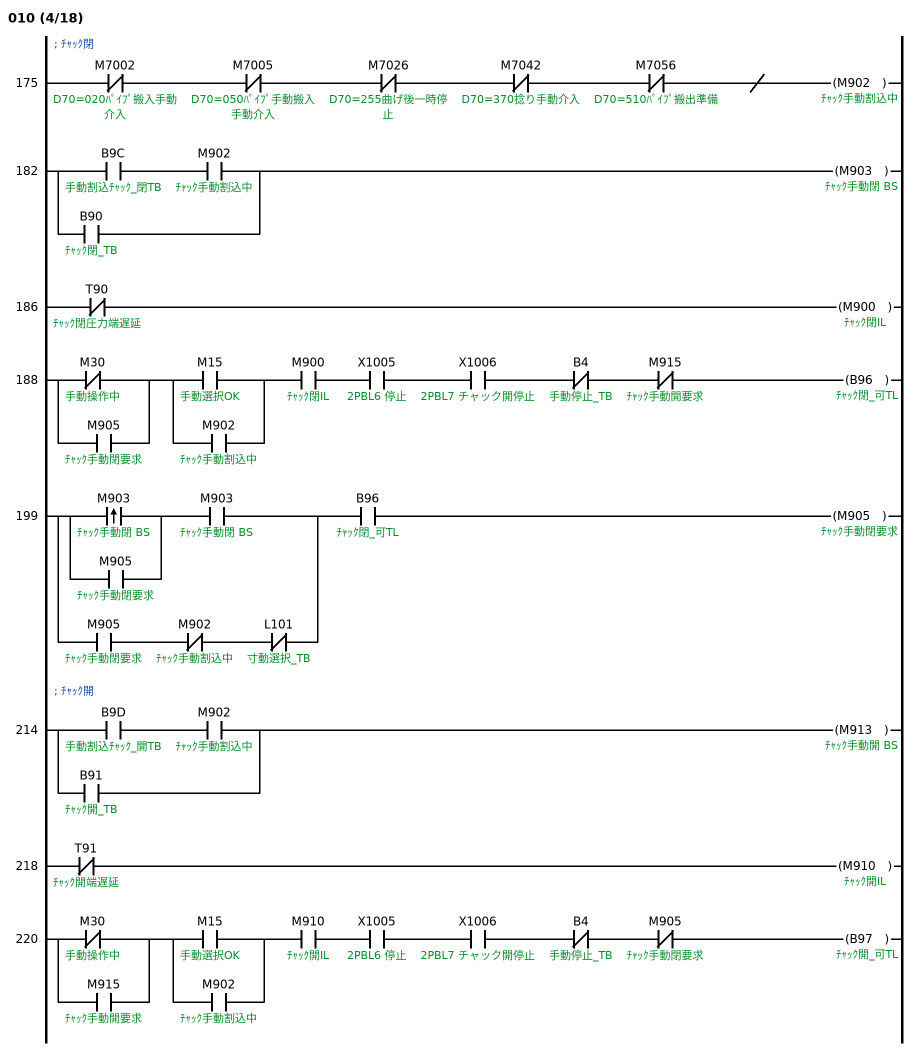
; ﾁｬｯｸ閉
175   LDI     M7002  ; D70=020ﾊﾟｲﾌﾟ搬入手動介入
      ANI     M7005  ; D70=050ﾊﾟｲﾌﾟ手動搬入手動介入
      ANI     M7026  ; D70=255曲げ後一時停止
      ANI     M7042  ; D70=370捻り手動介入
      ANI     M7056  ; D70=510ﾊﾟｲﾌﾟ搬出準備
      INV
      OUT     M902  ; ﾁｬｯｸ手動割込中
182   LD      B9C  ; 手動割込ﾁｬｯｸ_閉TB
      AND     M902  ; ﾁｬｯｸ手動割込中
      OR      B90  ; ﾁｬｯｸ閉_TB
      OUT     M903  ; ﾁｬｯｸ手動閉 BS
186   LDI     T90  ; ﾁｬｯｸ閉圧力端遅延
      OUT     M900  ; ﾁｬｯｸ閉IL
188   LDI     M30  ; 手動操作中
      OR      M905  ; ﾁｬｯｸ手動閉要求
      LD      M15  ; 手動選択OK
      OR      M902  ; ﾁｬｯｸ手動割込中
      ANB
      AND     M900  ; ﾁｬｯｸ閉IL
      AND     X1005  ; 2PBL6 停止
      AND     X1006  ; 2PBL7 チャック開停止
      ANI     B4  ; 手動停止_TB
      ANI     M915  ; ﾁｬｯｸ手動開要求
      OUT     B96  ; ﾁｬｯｸ閉_可TL
199   LDP     M903  ; ﾁｬｯｸ手動閉 BS
      OR      M905  ; ﾁｬｯｸ手動閉要求
      AND     M903  ; ﾁｬｯｸ手動閉 BS
      LD      M905  ; ﾁｬｯｸ手動閉要求
      ANI     M902  ; ﾁｬｯｸ手動割込中
      ANI     L101  ; 寸動選択_TB
      ORB
      AND     B96  ; ﾁｬｯｸ閉_可TL
      OUT     M905  ; ﾁｬｯｸ手動閉要求
; ﾁｬｯｸ開
214   LD      B9D  ; 手動割込ﾁｬｯｸ_開TB
      AND     M902  ; ﾁｬｯｸ手動割込中
      OR      B91  ; ﾁｬｯｸ開_TB
      OUT     M913  ; ﾁｬｯｸ手動開 BS
218   LDI     T91  ; ﾁｬｯｸ開端遅延
      OUT     M910  ; ﾁｬｯｸ開IL
220   LDI     M30  ; 手動操作中
      OR      M915  ; ﾁｬｯｸ手動開要求
      LD      M15  ; 手動選択OK
      OR      M902  ; ﾁｬｯｸ手動割込中
      ANB
      AND     M910  ; ﾁｬｯｸ開IL
      AND     X1005  ; 2PBL6 停止
      AND     X1006  ; 2PBL7 チャック開停止
      ANI     B4  ; 手動停止_TB
      ANI     M905  ; ﾁｬｯｸ手動閉要求
      OUT     B97  ; ﾁｬｯｸ開_可TL
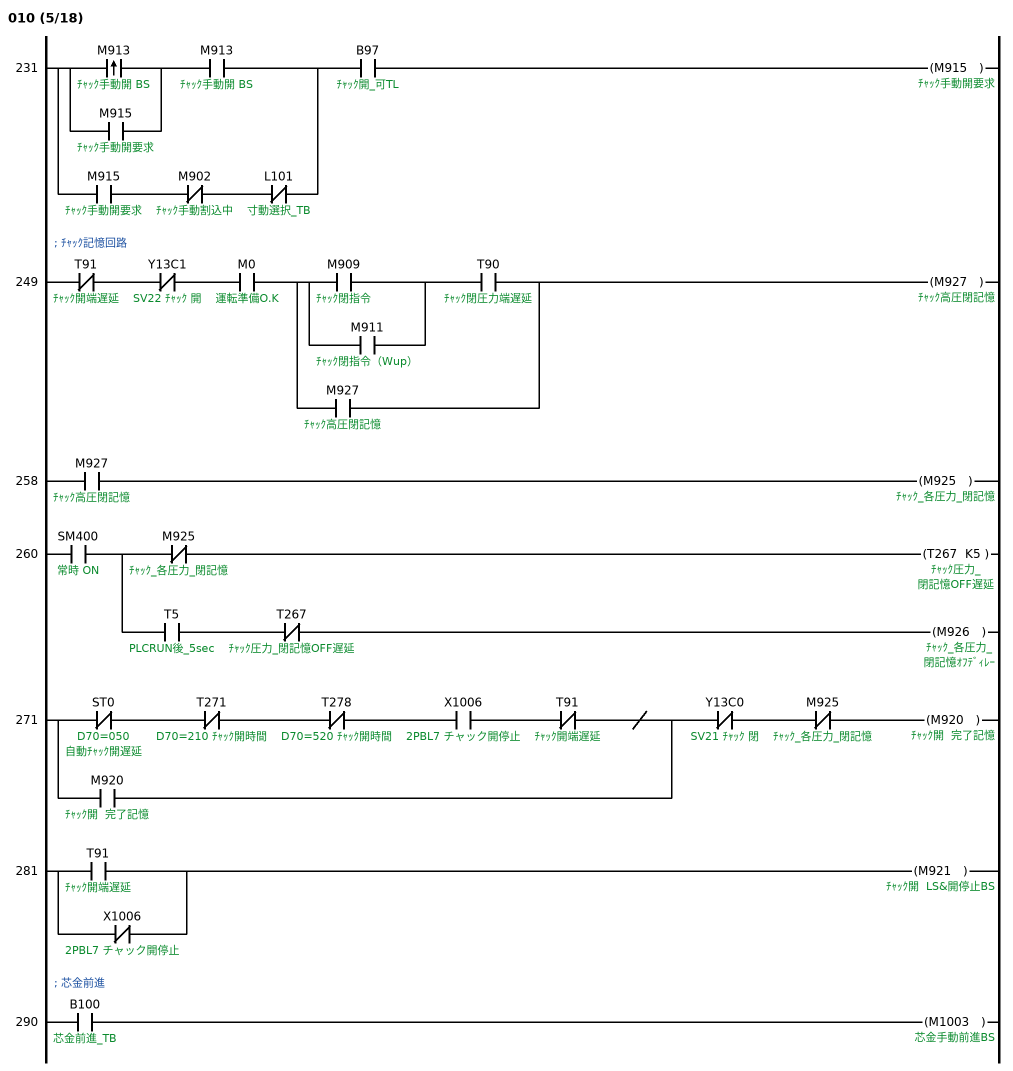
231   LDP     M913  ; ﾁｬｯｸ手動開 BS
      OR      M915  ; ﾁｬｯｸ手動開要求
      AND     M913  ; ﾁｬｯｸ手動開 BS
      LD      M915  ; ﾁｬｯｸ手動開要求
      ANI     M902  ; ﾁｬｯｸ手動割込中
      ANI     L101  ; 寸動選択_TB
      ORB
      AND     B97  ; ﾁｬｯｸ開_可TL
      OUT     M915  ; ﾁｬｯｸ手動開要求
; ﾁｬｯｸ記憶回路
249   LDI     T91  ; ﾁｬｯｸ開端遅延
      ANI     Y13C1  ; SV22 ﾁｬｯｸ 開
      AND     M0  ; 運転準備O.K
      LD      M909  ; ﾁｬｯｸ閉指令
      OR      M911  ; ﾁｬｯｸ閉指令（Wup）
      AND     T90  ; ﾁｬｯｸ閉圧力端遅延
      OR      M927  ; ﾁｬｯｸ高圧閉記憶
      ANB
      OUT     M927  ; ﾁｬｯｸ高圧閉記憶
258   LD      M927  ; ﾁｬｯｸ高圧閉記憶
      OUT     M925  ; ﾁｬｯｸ_各圧力_閉記憶
260   LD      SM400  ; 常時 ON
      MPS
      ANI     M925  ; ﾁｬｯｸ_各圧力_閉記憶
      OUT     T267 K5  ; ﾁｬｯｸ圧力_閉記憶OFF遅延
      MPP
      AND     T5  ; PLCRUN後_5sec
      ANI     T267  ; ﾁｬｯｸ圧力_閉記憶OFF遅延
      OUT     M926  ; ﾁｬｯｸ_各圧力_閉記憶ｵﾌﾃﾞｨﾚｰ
271   LDI     ST0  ; D70=050 自動ﾁｬｯｸ開遅延
      ANI     T271  ; D70=210 ﾁｬｯｸ開時間
      ANI     T278  ; D70=520 ﾁｬｯｸ開時間
      AND     X1006  ; 2PBL7 チャック開停止
      ANI     T91  ; ﾁｬｯｸ開端遅延
      INV
      OR      M920  ; ﾁｬｯｸ開  完了記憶
      ANI     Y13C0  ; SV21 ﾁｬｯｸ 閉
      ANI     M925  ; ﾁｬｯｸ_各圧力_閉記憶
      OUT     M920  ; ﾁｬｯｸ開  完了記憶
281   LD      T91  ; ﾁｬｯｸ開端遅延
      ORI     X1006  ; 2PBL7 チャック開停止
      OUT     M921  ; ﾁｬｯｸ開  LS&開停止BS
; 芯金前進
290   LD      B100  ; 芯金前進_TB
      OUT     M1003  ; 芯金手動前進BS
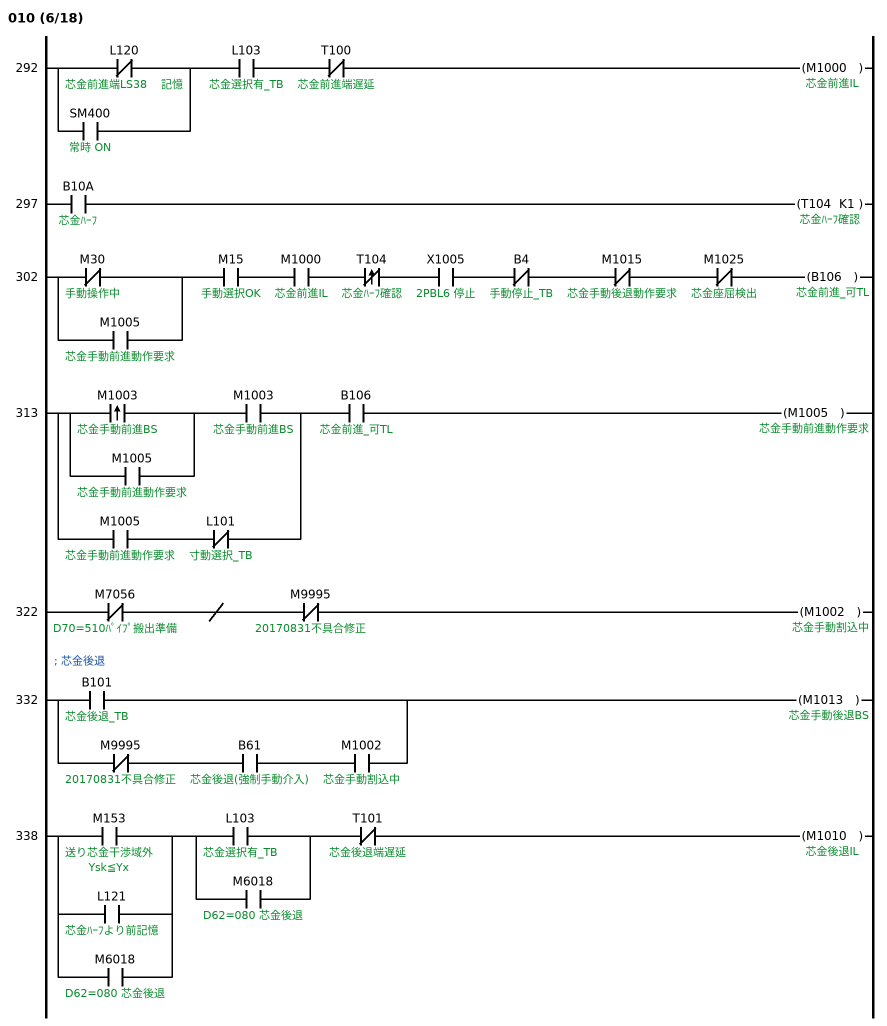
292   LDI     L120  ; 芯金前進端LS38    記憶
      OR      SM400  ; 常時 ON
      AND     L103  ; 芯金選択有_TB
      ANI     T100  ; 芯金前進端遅延
      OUT     M1000  ; 芯金前進IL
297   LD      B10A  ; 芯金ﾊｰﾌ
      OUT     T104 K1  ; 芯金ﾊｰﾌ確認
302   LDI     M30  ; 手動操作中
      OR      M1005  ; 芯金手動前進動作要求
      AND     M15  ; 手動選択OK
      AND     M1000  ; 芯金前進IL
      ANDPI   T104  ; 芯金ﾊｰﾌ確認
      AND     X1005  ; 2PBL6 停止
      ANI     B4  ; 手動停止_TB
      ANI     M1015  ; 芯金手動後退動作要求
      ANI     M1025  ; 芯金座屈検出
      OUT     B106  ; 芯金前進_可TL
313   LDP     M1003  ; 芯金手動前進BS
      OR      M1005  ; 芯金手動前進動作要求
      AND     M1003  ; 芯金手動前進BS
      LD      M1005  ; 芯金手動前進動作要求
      ANI     L101  ; 寸動選択_TB
      ORB
      AND     B106  ; 芯金前進_可TL
      OUT     M1005  ; 芯金手動前進動作要求
322   LDI     M7056  ; D70=510ﾊﾟｲﾌﾟ搬出準備
      INV
      ANI     M9995  ; 20170831不具合修正
      OUT     M1002  ; 芯金手動割込中
; 芯金後退
332   LD      B101  ; 芯金後退_TB
      LDI     M9995  ; 20170831不具合修正
      AND     B61  ; 芯金後退(強制手動介入)
      AND     M1002  ; 芯金手動割込中
      ORB
      OUT     M1013  ; 芯金手動後退BS
338   LD      M153  ; 送り芯金干渉域外 Ysk≦Yx
      OR      L121  ; 芯金ﾊｰﾌより前記憶
      OR      M6018  ; D62=080 芯金後退
      LD      L103  ; 芯金選択有_TB
      OR      M6018  ; D62=080 芯金後退
      ANB
      ANI     T101  ; 芯金後退端遅延
      OUT     M1010  ; 芯金後退IL
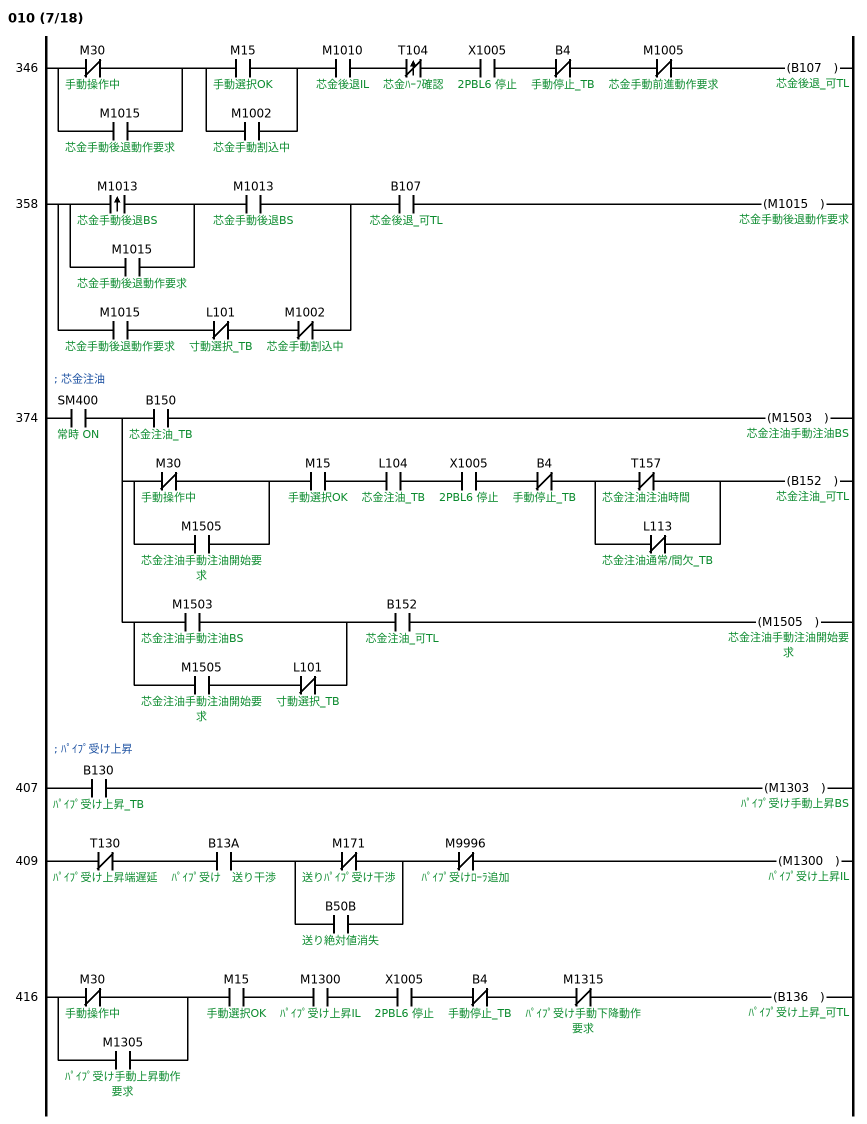
346   LDI     M30  ; 手動操作中
      OR      M1015  ; 芯金手動後退動作要求
      LD      M15  ; 手動選択OK
      OR      M1002  ; 芯金手動割込中
      ANB
      AND     M1010  ; 芯金後退IL
      ANDPI   T104  ; 芯金ﾊｰﾌ確認
      AND     X1005  ; 2PBL6 停止
      ANI     B4  ; 手動停止_TB
      ANI     M1005  ; 芯金手動前進動作要求
      OUT     B107  ; 芯金後退_可TL
358   LDP     M1013  ; 芯金手動後退BS
      OR      M1015  ; 芯金手動後退動作要求
      AND     M1013  ; 芯金手動後退BS
      LD      M1015  ; 芯金手動後退動作要求
      ANI     L101  ; 寸動選択_TB
      ANI     M1002  ; 芯金手動割込中
      ORB
      AND     B107  ; 芯金後退_可TL
      OUT     M1015  ; 芯金手動後退動作要求
; 芯金注油
374   LD      SM400  ; 常時 ON
      MPS
      AND     B150  ; 芯金注油_TB
      OUT     M1503  ; 芯金注油手動注油BS
      MRD
      LDI     M30  ; 手動操作中
      OR      M1505  ; 芯金注油手動注油開始要求
      ANB
      AND     M15  ; 手動選択OK
      AND     L104  ; 芯金注油_TB
      AND     X1005  ; 2PBL6 停止
      ANI     B4  ; 手動停止_TB
      LDI     T157  ; 芯金注油注油時間
      ORI     L113  ; 芯金注油通常/間欠_TB
      ANB
      OUT     B152  ; 芯金注油_可TL
      MPP
      LD      M1503  ; 芯金注油手動注油BS
      LD      M1505  ; 芯金注油手動注油開始要求
      ANI     L101  ; 寸動選択_TB
      ORB
      ANB
      AND     B152  ; 芯金注油_可TL
      OUT     M1505  ; 芯金注油手動注油開始要求
; ﾊﾟｲﾌﾟ受け上昇
407   LD      B130  ; ﾊﾟｲﾌﾟ受け上昇_TB
      OUT     M1303  ; ﾊﾟｲﾌﾟ受け手動上昇BS
409   LDI     T130  ; ﾊﾟｲﾌﾟ受け上昇端遅延
      AND     B13A  ; ﾊﾟｲﾌﾟ受け　送り干渉
      LDI     M171  ; 送りﾊﾟｲﾌﾟ受け干渉
      OR      B50B  ; 送り絶対値消失
      ANB
      ANI     M9996  ; ﾊﾟｲﾌﾟ受けﾛｰﾗ追加
      OUT     M1300  ; ﾊﾟｲﾌﾟ受け上昇IL
416   LDI     M30  ; 手動操作中
      OR      M1305  ; ﾊﾟｲﾌﾟ受け手動上昇動作要求
      AND     M15  ; 手動選択OK
      AND     M1300  ; ﾊﾟｲﾌﾟ受け上昇IL
      AND     X1005  ; 2PBL6 停止
      ANI     B4  ; 手動停止_TB
      ANI     M1315  ; ﾊﾟｲﾌﾟ受け手動下降動作要求
      OUT     B136  ; ﾊﾟｲﾌﾟ受け上昇_可TL
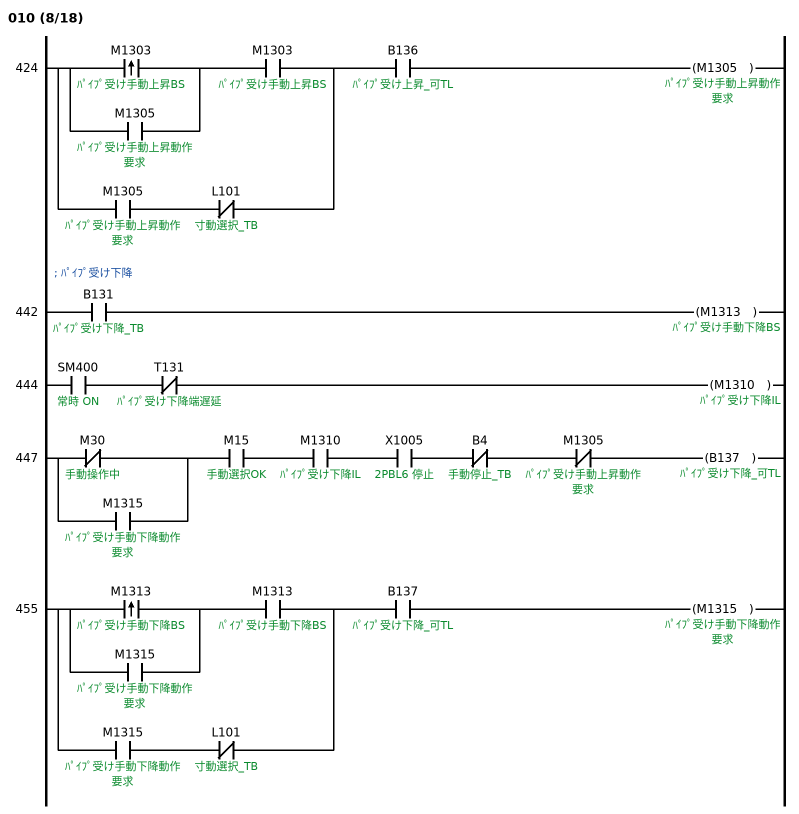
424   LDP     M1303  ; ﾊﾟｲﾌﾟ受け手動上昇BS
      OR      M1305  ; ﾊﾟｲﾌﾟ受け手動上昇動作要求
      AND     M1303  ; ﾊﾟｲﾌﾟ受け手動上昇BS
      LD      M1305  ; ﾊﾟｲﾌﾟ受け手動上昇動作要求
      ANI     L101  ; 寸動選択_TB
      ORB
      AND     B136  ; ﾊﾟｲﾌﾟ受け上昇_可TL
      OUT     M1305  ; ﾊﾟｲﾌﾟ受け手動上昇動作要求
; ﾊﾟｲﾌﾟ受け下降
442   LD      B131  ; ﾊﾟｲﾌﾟ受け下降_TB
      OUT     M1313  ; ﾊﾟｲﾌﾟ受け手動下降BS
444   LD      SM400  ; 常時 ON
      ANI     T131  ; ﾊﾟｲﾌﾟ受け下降端遅延
      OUT     M1310  ; ﾊﾟｲﾌﾟ受け下降IL
447   LDI     M30  ; 手動操作中
      OR      M1315  ; ﾊﾟｲﾌﾟ受け手動下降動作要求
      AND     M15  ; 手動選択OK
      AND     M1310  ; ﾊﾟｲﾌﾟ受け下降IL
      AND     X1005  ; 2PBL6 停止
      ANI     B4  ; 手動停止_TB
      ANI     M1305  ; ﾊﾟｲﾌﾟ受け手動上昇動作要求
      OUT     B137  ; ﾊﾟｲﾌﾟ受け下降_可TL
455   LDP     M1313  ; ﾊﾟｲﾌﾟ受け手動下降BS
      OR      M1315  ; ﾊﾟｲﾌﾟ受け手動下降動作要求
      AND     M1313  ; ﾊﾟｲﾌﾟ受け手動下降BS
      LD      M1315  ; ﾊﾟｲﾌﾟ受け手動下降動作要求
      ANI     L101  ; 寸動選択_TB
      ORB
      AND     B137  ; ﾊﾟｲﾌﾟ受け下降_可TL
      OUT     M1315  ; ﾊﾟｲﾌﾟ受け手動下降動作要求
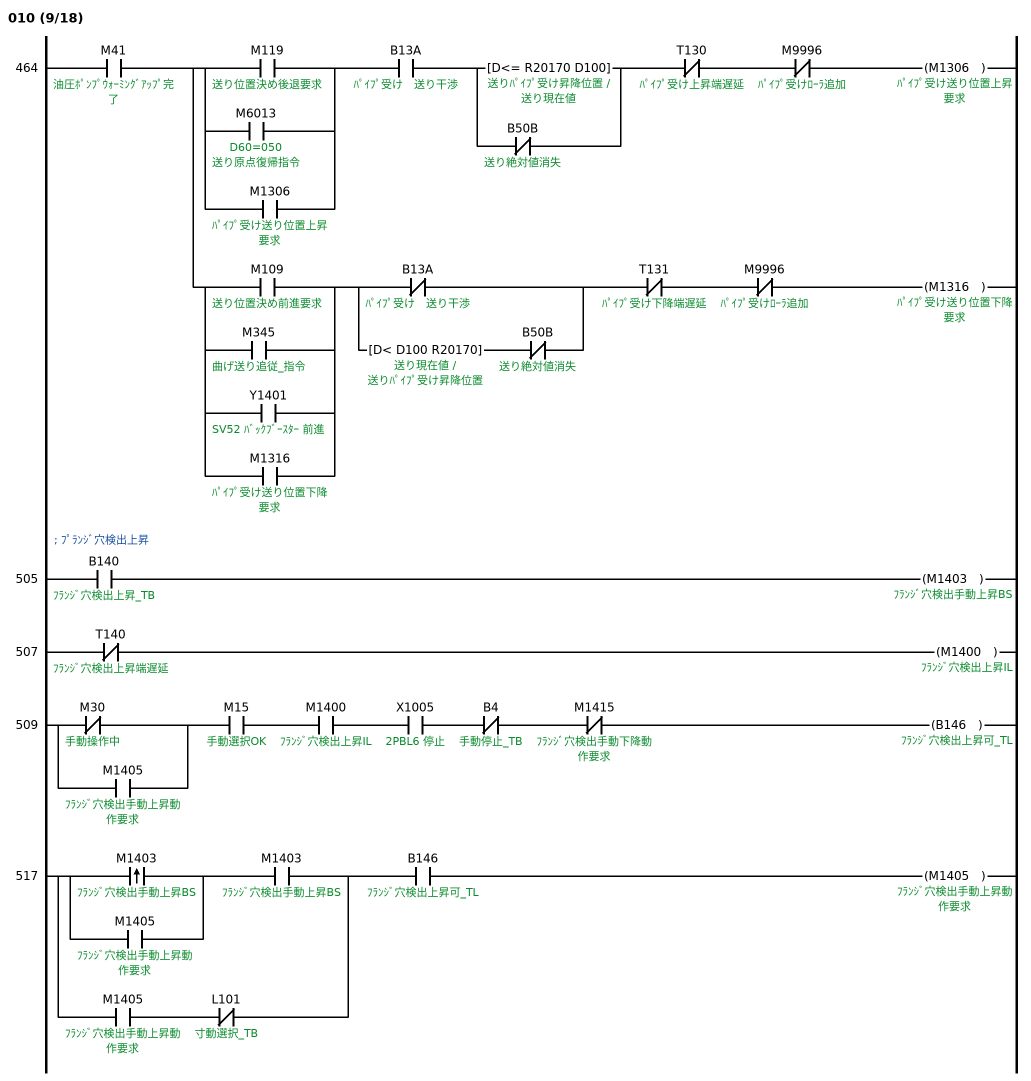
464   LD      M41  ; 油圧ﾎﾟﾝﾌﾟｳｫｰﾐﾝｸﾞｱｯﾌﾟ完了
      MPS
      LD      M119  ; 送り位置決め後退要求
      OR      M6013  ; D60=050 送り原点復帰指令
      OR      M1306  ; ﾊﾟｲﾌﾟ受け送り位置上昇要求
      ANB
      AND     B13A  ; ﾊﾟｲﾌﾟ受け　送り干渉
      LDD<=   R20170 D100  ; 送りﾊﾟｲﾌﾟ受け昇降位置 / 送り現在値
      ORI     B50B  ; 送り絶対値消失
      ANB
      ANI     T130  ; ﾊﾟｲﾌﾟ受け上昇端遅延
      ANI     M9996  ; ﾊﾟｲﾌﾟ受けﾛｰﾗ追加
      OUT     M1306  ; ﾊﾟｲﾌﾟ受け送り位置上昇要求
      MPP
      LD      M109  ; 送り位置決め前進要求
      OR      M345  ; 曲げ送り追従_指令
      OR      Y1401  ; SV52 ﾊﾞｯｸﾌﾞｰｽﾀｰ 前進
      OR      M1316  ; ﾊﾟｲﾌﾟ受け送り位置下降要求
      ANB
      LDI     B13A  ; ﾊﾟｲﾌﾟ受け　送り干渉
      LDD<    D100 R20170  ; 送り現在値 / 送りﾊﾟｲﾌﾟ受け昇降位置
      ANI     B50B  ; 送り絶対値消失
      ORB
      ANB
      ANI     T131  ; ﾊﾟｲﾌﾟ受け下降端遅延
      ANI     M9996  ; ﾊﾟｲﾌﾟ受けﾛｰﾗ追加
      OUT     M1316  ; ﾊﾟｲﾌﾟ受け送り位置下降要求
; ﾌﾟﾗﾝｼﾞ穴検出上昇
505   LD      B140  ; ﾌﾗﾝｼﾞ穴検出上昇_TB
      OUT     M1403  ; ﾌﾗﾝｼﾞ穴検出手動上昇BS
507   LDI     T140  ; ﾌﾗﾝｼﾞ穴検出上昇端遅延
      OUT     M1400  ; ﾌﾗﾝｼﾞ穴検出上昇IL
509   LDI     M30  ; 手動操作中
      OR      M1405  ; ﾌﾗﾝｼﾞ穴検出手動上昇動作要求
      AND     M15  ; 手動選択OK
      AND     M1400  ; ﾌﾗﾝｼﾞ穴検出上昇IL
      AND     X1005  ; 2PBL6 停止
      ANI     B4  ; 手動停止_TB
      ANI     M1415  ; ﾌﾗﾝｼﾞ穴検出手動下降動作要求
      OUT     B146  ; ﾌﾗﾝｼﾞ穴検出上昇可_TL
517   LDP     M1403  ; ﾌﾗﾝｼﾞ穴検出手動上昇BS
      OR      M1405  ; ﾌﾗﾝｼﾞ穴検出手動上昇動作要求
      AND     M1403  ; ﾌﾗﾝｼﾞ穴検出手動上昇BS
      LD      M1405  ; ﾌﾗﾝｼﾞ穴検出手動上昇動作要求
      ANI     L101  ; 寸動選択_TB
      ORB
      AND     B146  ; ﾌﾗﾝｼﾞ穴検出上昇可_TL
      OUT     M1405  ; ﾌﾗﾝｼﾞ穴検出手動上昇動作要求
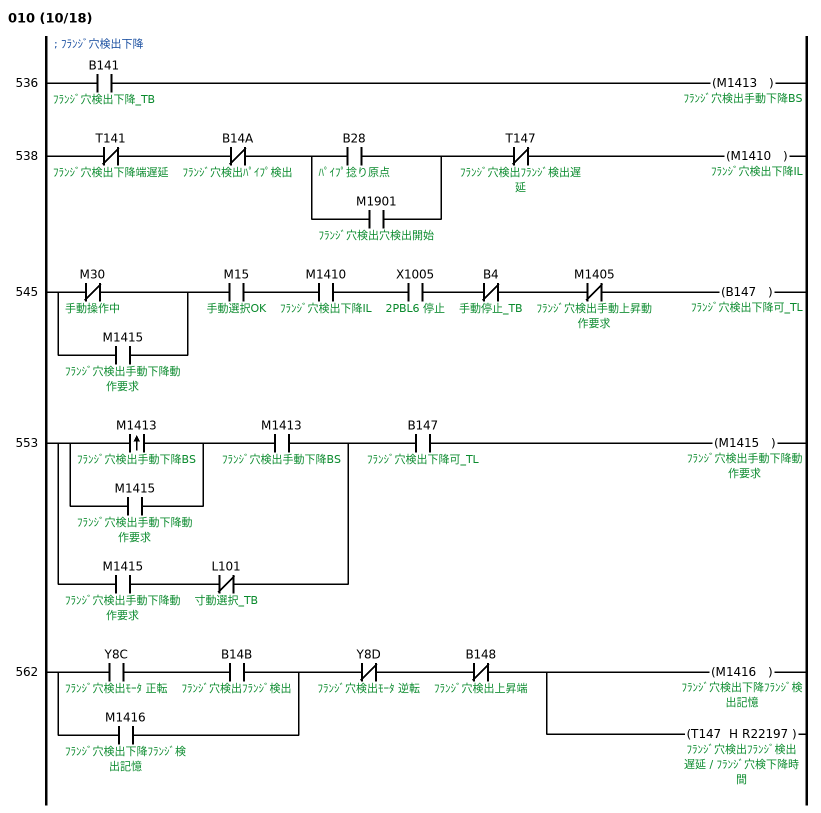
; ﾌﾗﾝｼﾞ穴検出下降
536   LD      B141  ; ﾌﾗﾝｼﾞ穴検出下降_TB
      OUT     M1413  ; ﾌﾗﾝｼﾞ穴検出手動下降BS
538   LDI     T141  ; ﾌﾗﾝｼﾞ穴検出下降端遅延
      ANI     B14A  ; ﾌﾗﾝｼﾞ穴検出ﾊﾟｲﾌﾟ検出
      LD      B28  ; ﾊﾟｲﾌﾟ捻り原点
      OR      M1901  ; ﾌﾗﾝｼﾞ穴検出穴検出開始
      ANB
      ANI     T147  ; ﾌﾗﾝｼﾞ穴検出ﾌﾗﾝｼﾞ検出遅延
      OUT     M1410  ; ﾌﾗﾝｼﾞ穴検出下降IL
545   LDI     M30  ; 手動操作中
      OR      M1415  ; ﾌﾗﾝｼﾞ穴検出手動下降動作要求
      AND     M15  ; 手動選択OK
      AND     M1410  ; ﾌﾗﾝｼﾞ穴検出下降IL
      AND     X1005  ; 2PBL6 停止
      ANI     B4  ; 手動停止_TB
      ANI     M1405  ; ﾌﾗﾝｼﾞ穴検出手動上昇動作要求
      OUT     B147  ; ﾌﾗﾝｼﾞ穴検出下降可_TL
553   LDP     M1413  ; ﾌﾗﾝｼﾞ穴検出手動下降BS
      OR      M1415  ; ﾌﾗﾝｼﾞ穴検出手動下降動作要求
      AND     M1413  ; ﾌﾗﾝｼﾞ穴検出手動下降BS
      LD      M1415  ; ﾌﾗﾝｼﾞ穴検出手動下降動作要求
      ANI     L101  ; 寸動選択_TB
      ORB
      AND     B147  ; ﾌﾗﾝｼﾞ穴検出下降可_TL
      OUT     M1415  ; ﾌﾗﾝｼﾞ穴検出手動下降動作要求
562   LD      Y8C  ; ﾌﾗﾝｼﾞ穴検出ﾓｰﾀ 正転
      AND     B14B  ; ﾌﾗﾝｼﾞ穴検出ﾌﾗﾝｼﾞ検出
      OR      M1416  ; ﾌﾗﾝｼﾞ穴検出下降ﾌﾗﾝｼﾞ検出記憶
      ANI     Y8D  ; ﾌﾗﾝｼﾞ穴検出ﾓｰﾀ 逆転
      ANI     B148  ; ﾌﾗﾝｼﾞ穴検出上昇端
      OUT     M1416  ; ﾌﾗﾝｼﾞ穴検出下降ﾌﾗﾝｼﾞ検出記憶
      OUTH    T147 R22197  ; ﾌﾗﾝｼﾞ穴検出ﾌﾗﾝｼﾞ検出遅延 / ﾌﾗﾝｼﾞ穴検下降時間
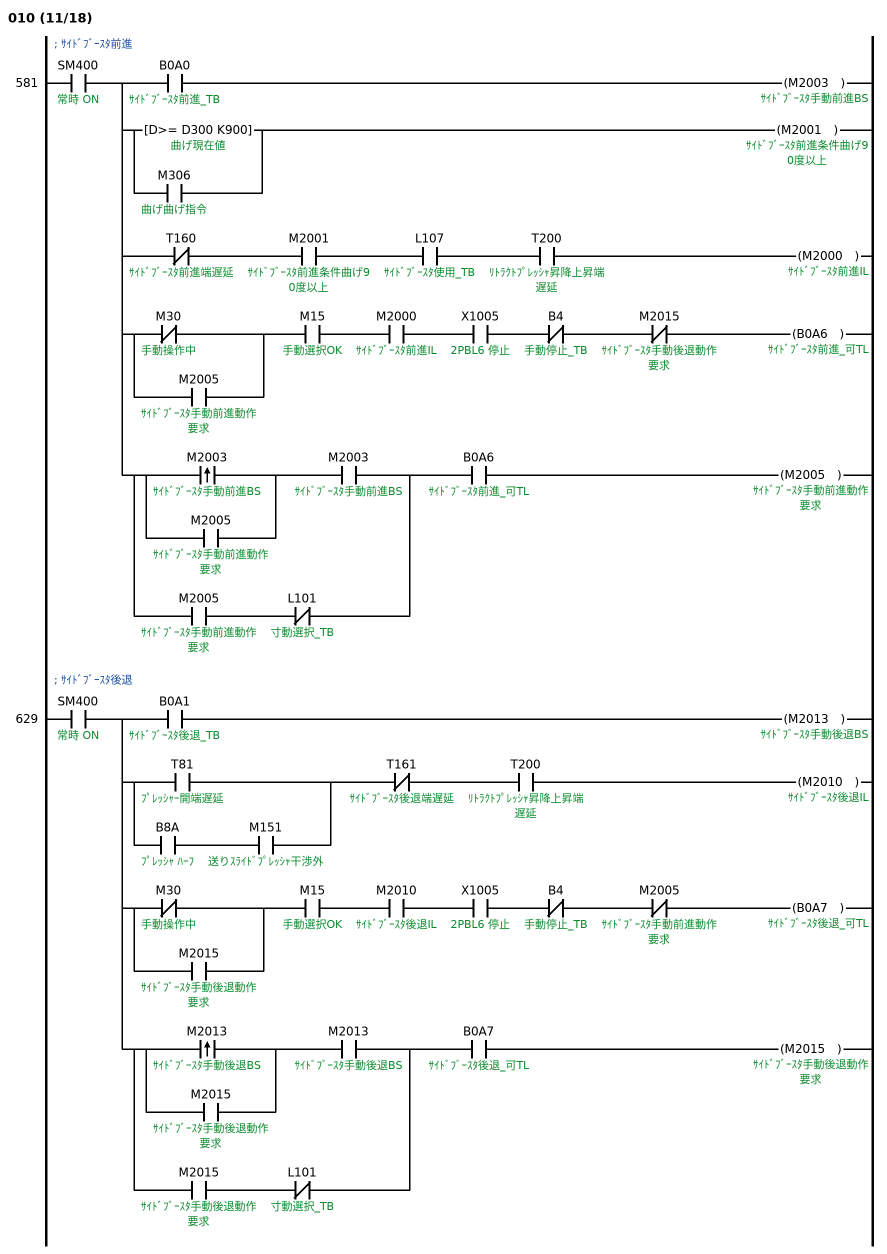
; ｻｲﾄﾞﾌﾞｰｽﾀ前進
581   LD      SM400  ; 常時 ON
      MPS
      AND     B0A0  ; ｻｲﾄﾞﾌﾞｰｽﾀ前進_TB
      OUT     M2003  ; ｻｲﾄﾞﾌﾞｰｽﾀ手動前進BS
      MRD
      LDD>=   D300 K900  ; 曲げ現在値
      OR      M306  ; 曲げ曲げ指令
      ANB
      OUT     M2001  ; ｻｲﾄﾞﾌﾞｰｽﾀ前進条件曲げ90度以上
      MRD
      ANI     T160  ; ｻｲﾄﾞﾌﾞｰｽﾀ前進端遅延
      AND     M2001  ; ｻｲﾄﾞﾌﾞｰｽﾀ前進条件曲げ90度以上
      AND     L107  ; ｻｲﾄﾞﾌﾞｰｽﾀ使用_TB
      AND     T200  ; ﾘﾄﾗｸﾄﾌﾟﾚｯｼｬ昇降上昇端遅延
      OUT     M2000  ; ｻｲﾄﾞﾌﾞｰｽﾀ前進IL
      MRD
      LDI     M30  ; 手動操作中
      OR      M2005  ; ｻｲﾄﾞﾌﾞｰｽﾀ手動前進動作要求
      ANB
      AND     M15  ; 手動選択OK
      AND     M2000  ; ｻｲﾄﾞﾌﾞｰｽﾀ前進IL
      AND     X1005  ; 2PBL6 停止
      ANI     B4  ; 手動停止_TB
      ANI     M2015  ; ｻｲﾄﾞﾌﾞｰｽﾀ手動後退動作要求
      OUT     B0A6  ; ｻｲﾄﾞﾌﾞｰｽﾀ前進_可TL
      MPP
      LDP     M2003  ; ｻｲﾄﾞﾌﾞｰｽﾀ手動前進BS
      OR      M2005  ; ｻｲﾄﾞﾌﾞｰｽﾀ手動前進動作要求
      AND     M2003  ; ｻｲﾄﾞﾌﾞｰｽﾀ手動前進BS
      LD      M2005  ; ｻｲﾄﾞﾌﾞｰｽﾀ手動前進動作要求
      ANI     L101  ; 寸動選択_TB
      ORB
      ANB
      AND     B0A6  ; ｻｲﾄﾞﾌﾞｰｽﾀ前進_可TL
      OUT     M2005  ; ｻｲﾄﾞﾌﾞｰｽﾀ手動前進動作要求
; ｻｲﾄﾞﾌﾞｰｽﾀ後退
629   LD      SM400  ; 常時 ON
      MPS
      AND     B0A1  ; ｻｲﾄﾞﾌﾞｰｽﾀ後退_TB
      OUT     M2013  ; ｻｲﾄﾞﾌﾞｰｽﾀ手動後退BS
      MRD
      LD      T81  ; ﾌﾟﾚｯｼｬｰ開端遅延
      LD      B8A  ; ﾌﾟﾚｯｼｬ ﾊｰﾌ
      AND     M151  ; 送りｽﾗｲﾄﾞﾌﾟﾚｯｼｬ干渉外
      ORB
      ANB
      ANI     T161  ; ｻｲﾄﾞﾌﾞｰｽﾀ後退端遅延
      AND     T200  ; ﾘﾄﾗｸﾄﾌﾟﾚｯｼｬ昇降上昇端遅延
      OUT     M2010  ; ｻｲﾄﾞﾌﾞｰｽﾀ後退IL
      MRD
      LDI     M30  ; 手動操作中
      OR      M2015  ; ｻｲﾄﾞﾌﾞｰｽﾀ手動後退動作要求
      ANB
      AND     M15  ; 手動選択OK
      AND     M2010  ; ｻｲﾄﾞﾌﾞｰｽﾀ後退IL
      AND     X1005  ; 2PBL6 停止
      ANI     B4  ; 手動停止_TB
      ANI     M2005  ; ｻｲﾄﾞﾌﾞｰｽﾀ手動前進動作要求
      OUT     B0A7  ; ｻｲﾄﾞﾌﾞｰｽﾀ後退_可TL
      MPP
      LDP     M2013  ; ｻｲﾄﾞﾌﾞｰｽﾀ手動後退BS
      OR      M2015  ; ｻｲﾄﾞﾌﾞｰｽﾀ手動後退動作要求
      AND     M2013  ; ｻｲﾄﾞﾌﾞｰｽﾀ手動後退BS
      LD      M2015  ; ｻｲﾄﾞﾌﾞｰｽﾀ手動後退動作要求
      ANI     L101  ; 寸動選択_TB
      ORB
      ANB
      AND     B0A7  ; ｻｲﾄﾞﾌﾞｰｽﾀ後退_可TL
      OUT     M2015  ; ｻｲﾄﾞﾌﾞｰｽﾀ手動後退動作要求
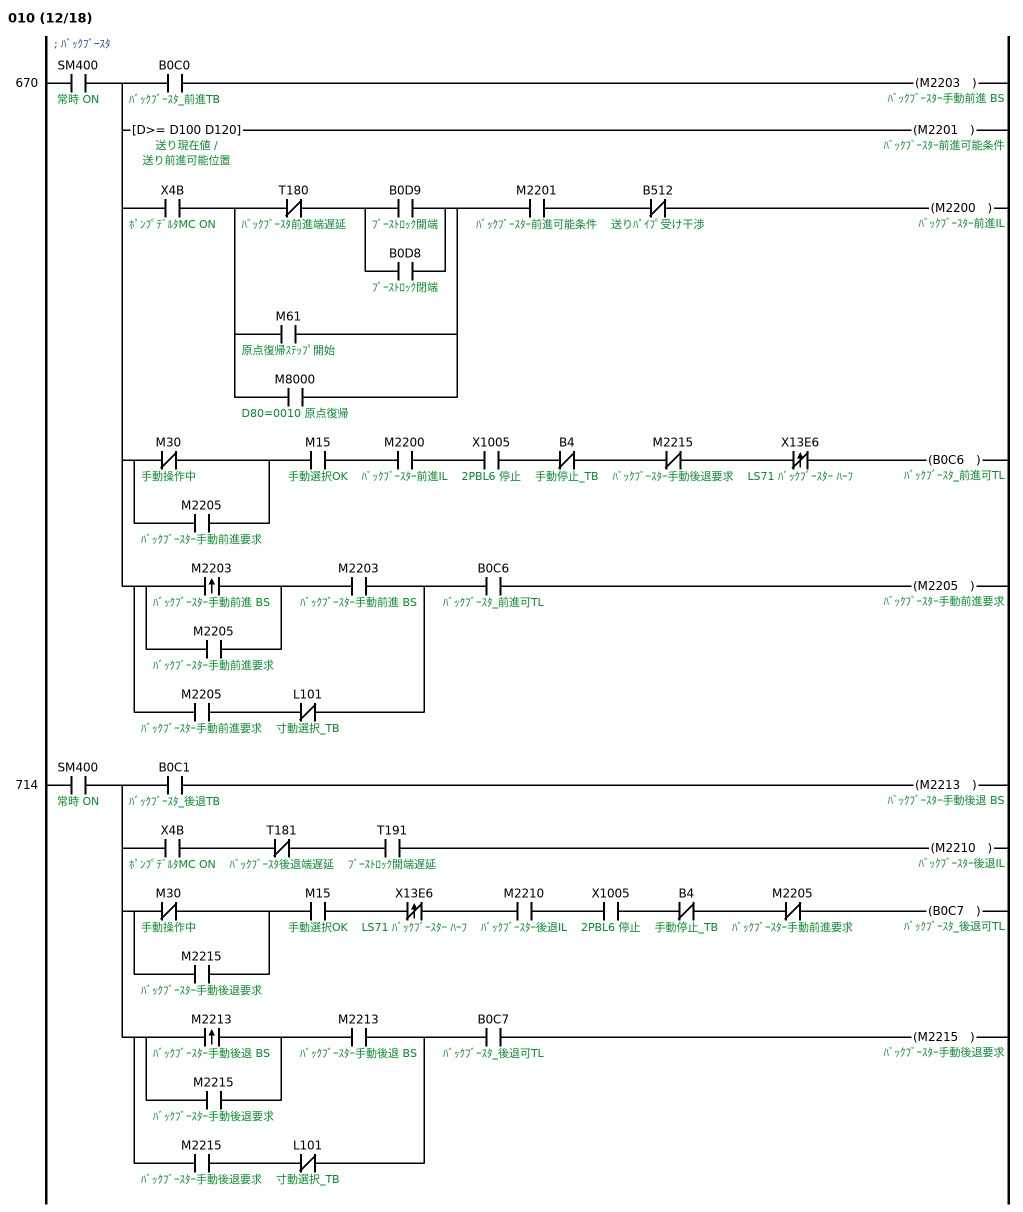
; ﾊﾞｯｸﾌﾞｰｽﾀ
670   LD      SM400  ; 常時 ON
      MPS
      AND     B0C0  ; ﾊﾞｯｸﾌﾞｰｽﾀ_前進TB
      OUT     M2203  ; ﾊﾞｯｸﾌﾞｰｽﾀｰ手動前進 BS
      MRD
      ANDD>=  D100 D120  ; 送り現在値 / 送り前進可能位置
      OUT     M2201  ; ﾊﾞｯｸﾌﾞｰｽﾀｰ前進可能条件
      MRD
      AND     X4B  ; ﾎﾟﾝﾌﾟﾃﾞﾙﾀMC ON
      LDI     T180  ; ﾊﾞｯｸﾌﾞｰｽﾀ前進端遅延
      LD      B0D9  ; ﾌﾞｰｽﾄﾛｯｸ開端
      OR      B0D8  ; ﾌﾞｰｽﾄﾛｯｸ閉端
      ANB
      OR      M61  ; 原点復帰ｽﾃｯﾌﾟ開始
      OR      M8000  ; D80=0010 原点復帰
      ANB
      AND     M2201  ; ﾊﾞｯｸﾌﾞｰｽﾀｰ前進可能条件
      ANI     B512  ; 送りﾊﾟｲﾌﾟ受け干渉
      OUT     M2200  ; ﾊﾞｯｸﾌﾞｰｽﾀｰ前進IL
      MRD
      LDI     M30  ; 手動操作中
      OR      M2205  ; ﾊﾞｯｸﾌﾞｰｽﾀｰ手動前進要求
      ANB
      AND     M15  ; 手動選択OK
      AND     M2200  ; ﾊﾞｯｸﾌﾞｰｽﾀｰ前進IL
      AND     X1005  ; 2PBL6 停止
      ANI     B4  ; 手動停止_TB
      ANI     M2215  ; ﾊﾞｯｸﾌﾞｰｽﾀｰ手動後退要求
      ANDPI   X13E6  ; LS71 ﾊﾞｯｸﾌﾞｰｽﾀｰ ﾊｰﾌ
      OUT     B0C6  ; ﾊﾞｯｸﾌﾞｰｽﾀ_前進可TL
      MPP
      LDP     M2203  ; ﾊﾞｯｸﾌﾞｰｽﾀｰ手動前進 BS
      OR      M2205  ; ﾊﾞｯｸﾌﾞｰｽﾀｰ手動前進要求
      AND     M2203  ; ﾊﾞｯｸﾌﾞｰｽﾀｰ手動前進 BS
      LD      M2205  ; ﾊﾞｯｸﾌﾞｰｽﾀｰ手動前進要求
      ANI     L101  ; 寸動選択_TB
      ORB
      ANB
      AND     B0C6  ; ﾊﾞｯｸﾌﾞｰｽﾀ_前進可TL
      OUT     M2205  ; ﾊﾞｯｸﾌﾞｰｽﾀｰ手動前進要求
714   LD      SM400  ; 常時 ON
      MPS
      AND     B0C1  ; ﾊﾞｯｸﾌﾞｰｽﾀ_後退TB
      OUT     M2213  ; ﾊﾞｯｸﾌﾞｰｽﾀｰ手動後退 BS
      MRD
      AND     X4B  ; ﾎﾟﾝﾌﾟﾃﾞﾙﾀMC ON
      ANI     T181  ; ﾊﾞｯｸﾌﾞｰｽﾀ後退端遅延
      AND     T191  ; ﾌﾞｰｽﾄﾛｯｸ開端遅延
      OUT     M2210  ; ﾊﾞｯｸﾌﾞｰｽﾀｰ後退IL
      MRD
      LDI     M30  ; 手動操作中
      OR      M2215  ; ﾊﾞｯｸﾌﾞｰｽﾀｰ手動後退要求
      ANB
      AND     M15  ; 手動選択OK
      ANDPI   X13E6  ; LS71 ﾊﾞｯｸﾌﾞｰｽﾀｰ ﾊｰﾌ
      AND     M2210  ; ﾊﾞｯｸﾌﾞｰｽﾀｰ後退IL
      AND     X1005  ; 2PBL6 停止
      ANI     B4  ; 手動停止_TB
      ANI     M2205  ; ﾊﾞｯｸﾌﾞｰｽﾀｰ手動前進要求
      OUT     B0C7  ; ﾊﾞｯｸﾌﾞｰｽﾀ_後退可TL
      MPP
      LDP     M2213  ; ﾊﾞｯｸﾌﾞｰｽﾀｰ手動後退 BS
      OR      M2215  ; ﾊﾞｯｸﾌﾞｰｽﾀｰ手動後退要求
      AND     M2213  ; ﾊﾞｯｸﾌﾞｰｽﾀｰ手動後退 BS
      LD      M2215  ; ﾊﾞｯｸﾌﾞｰｽﾀｰ手動後退要求
      ANI     L101  ; 寸動選択_TB
      ORB
      ANB
      AND     B0C7  ; ﾊﾞｯｸﾌﾞｰｽﾀ_後退可TL
      OUT     M2215  ; ﾊﾞｯｸﾌﾞｰｽﾀｰ手動後退要求
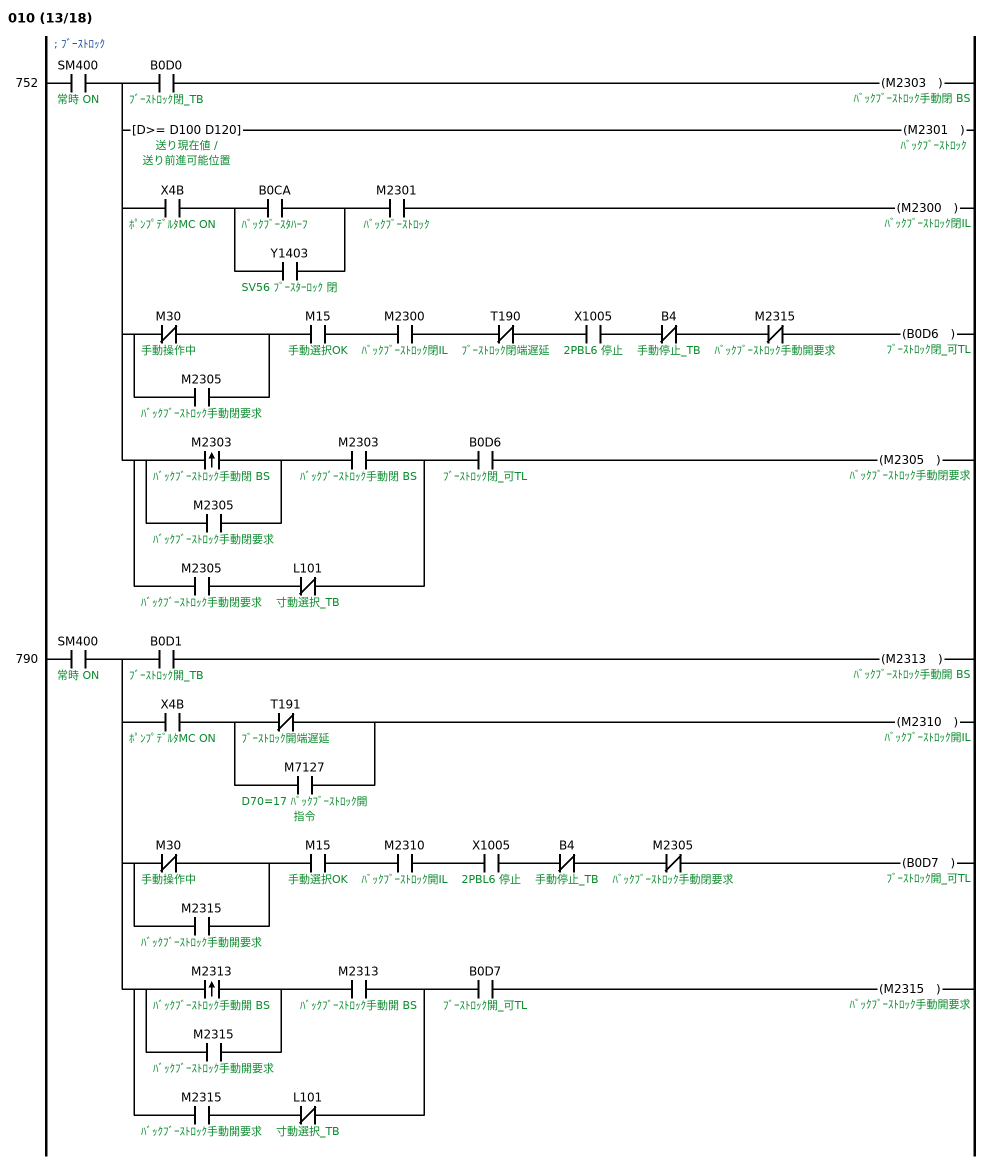
; ﾌﾞｰｽﾄﾛｯｸ
752   LD      SM400  ; 常時 ON
      MPS
      AND     B0D0  ; ﾌﾞｰｽﾄﾛｯｸ閉_TB
      OUT     M2303  ; ﾊﾞｯｸﾌﾞｰｽﾄﾛｯｸ手動閉 BS
      MRD
      ANDD>=  D100 D120  ; 送り現在値 / 送り前進可能位置
      OUT     M2301  ; ﾊﾞｯｸﾌﾞｰｽﾄﾛｯｸ
      MRD
      AND     X4B  ; ﾎﾟﾝﾌﾟﾃﾞﾙﾀMC ON
      LD      B0CA  ; ﾊﾞｯｸﾌﾞｰｽﾀﾊｰﾌ
      OR      Y1403  ; SV56 ﾌﾞｰｽﾀｰﾛｯｸ 閉
      ANB
      AND     M2301  ; ﾊﾞｯｸﾌﾞｰｽﾄﾛｯｸ
      OUT     M2300  ; ﾊﾞｯｸﾌﾞｰｽﾄﾛｯｸ閉IL
      MRD
      LDI     M30  ; 手動操作中
      OR      M2305  ; ﾊﾞｯｸﾌﾞｰｽﾄﾛｯｸ手動閉要求
      ANB
      AND     M15  ; 手動選択OK
      AND     M2300  ; ﾊﾞｯｸﾌﾞｰｽﾄﾛｯｸ閉IL
      ANI     T190  ; ﾌﾞｰｽﾄﾛｯｸ閉端遅延
      AND     X1005  ; 2PBL6 停止
      ANI     B4  ; 手動停止_TB
      ANI     M2315  ; ﾊﾞｯｸﾌﾞｰｽﾄﾛｯｸ手動開要求
      OUT     B0D6  ; ﾌﾞｰｽﾄﾛｯｸ閉_可TL
      MPP
      LDP     M2303  ; ﾊﾞｯｸﾌﾞｰｽﾄﾛｯｸ手動閉 BS
      OR      M2305  ; ﾊﾞｯｸﾌﾞｰｽﾄﾛｯｸ手動閉要求
      AND     M2303  ; ﾊﾞｯｸﾌﾞｰｽﾄﾛｯｸ手動閉 BS
      LD      M2305  ; ﾊﾞｯｸﾌﾞｰｽﾄﾛｯｸ手動閉要求
      ANI     L101  ; 寸動選択_TB
      ORB
      ANB
      AND     B0D6  ; ﾌﾞｰｽﾄﾛｯｸ閉_可TL
      OUT     M2305  ; ﾊﾞｯｸﾌﾞｰｽﾄﾛｯｸ手動閉要求
790   LD      SM400  ; 常時 ON
      MPS
      AND     B0D1  ; ﾌﾞｰｽﾄﾛｯｸ開_TB
      OUT     M2313  ; ﾊﾞｯｸﾌﾞｰｽﾄﾛｯｸ手動開 BS
      MRD
      AND     X4B  ; ﾎﾟﾝﾌﾟﾃﾞﾙﾀMC ON
      LDI     T191  ; ﾌﾞｰｽﾄﾛｯｸ開端遅延
      OR      M7127  ; D70=17 ﾊﾞｯｸﾌﾞｰｽﾄﾛｯｸ開指令
      ANB
      OUT     M2310  ; ﾊﾞｯｸﾌﾞｰｽﾄﾛｯｸ開IL
      MRD
      LDI     M30  ; 手動操作中
      OR      M2315  ; ﾊﾞｯｸﾌﾞｰｽﾄﾛｯｸ手動開要求
      ANB
      AND     M15  ; 手動選択OK
      AND     M2310  ; ﾊﾞｯｸﾌﾞｰｽﾄﾛｯｸ開IL
      AND     X1005  ; 2PBL6 停止
      ANI     B4  ; 手動停止_TB
      ANI     M2305  ; ﾊﾞｯｸﾌﾞｰｽﾄﾛｯｸ手動閉要求
      OUT     B0D7  ; ﾌﾞｰｽﾄﾛｯｸ開_可TL
      MPP
      LDP     M2313  ; ﾊﾞｯｸﾌﾞｰｽﾄﾛｯｸ手動開 BS
      OR      M2315  ; ﾊﾞｯｸﾌﾞｰｽﾄﾛｯｸ手動開要求
      AND     M2313  ; ﾊﾞｯｸﾌﾞｰｽﾄﾛｯｸ手動開 BS
      LD      M2315  ; ﾊﾞｯｸﾌﾞｰｽﾄﾛｯｸ手動開要求
      ANI     L101  ; 寸動選択_TB
      ORB
      ANB
      AND     B0D7  ; ﾌﾞｰｽﾄﾛｯｸ開_可TL
      OUT     M2315  ; ﾊﾞｯｸﾌﾞｰｽﾄﾛｯｸ手動開要求
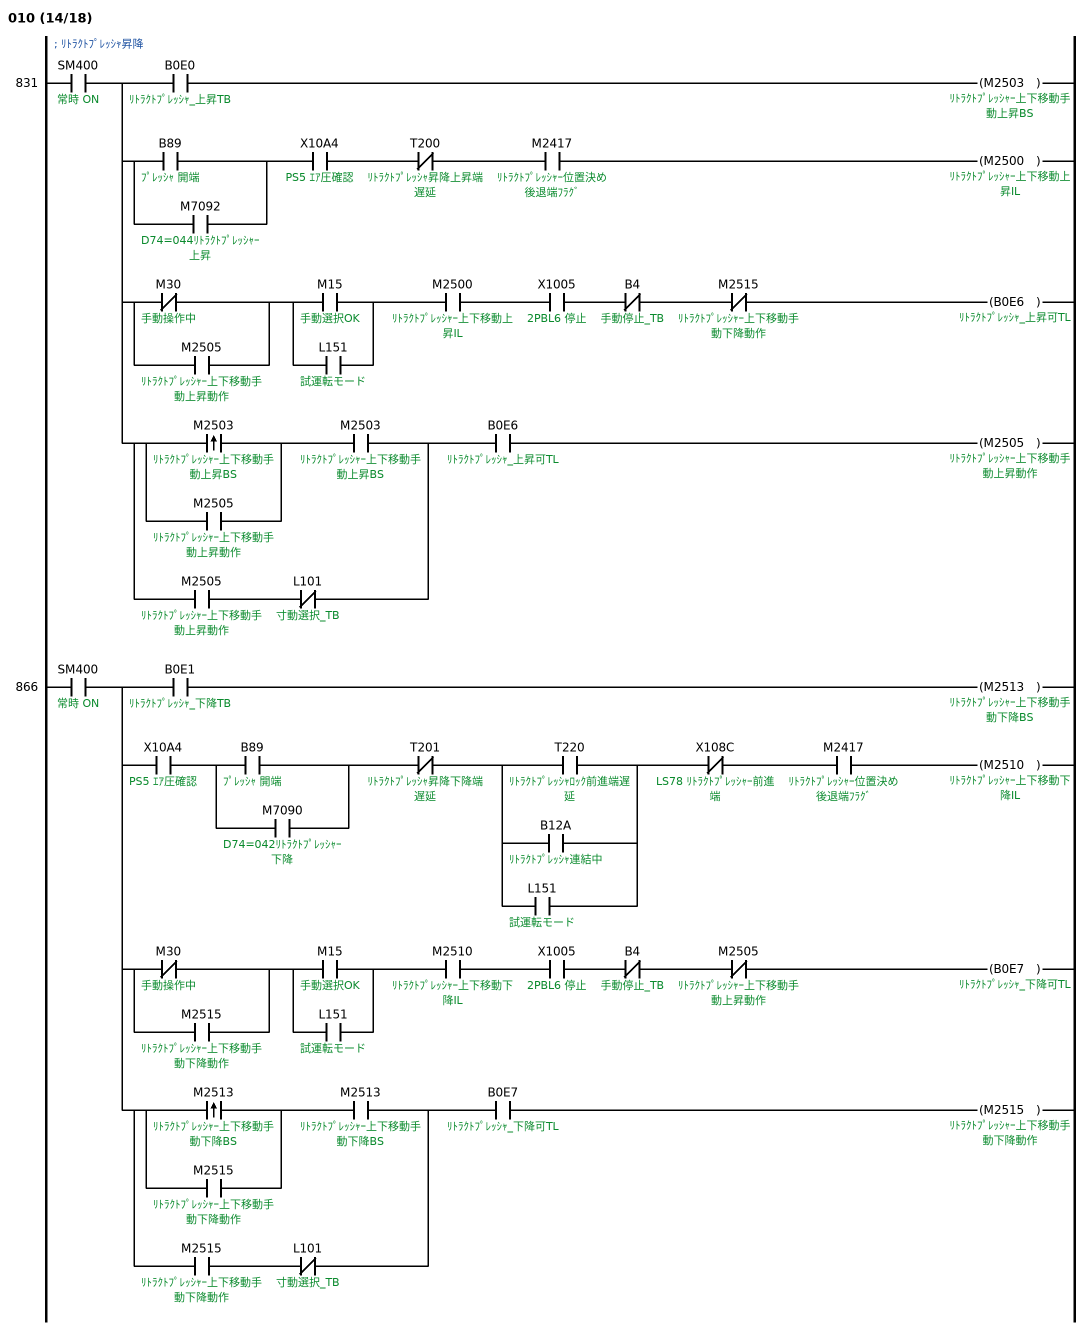
; ﾘﾄﾗｸﾄﾌﾟﾚｯｼｬ昇降
831   LD      SM400  ; 常時 ON
      MPS
      AND     B0E0  ; ﾘﾄﾗｸﾄﾌﾟﾚｯｼｬ_上昇TB
      OUT     M2503  ; ﾘﾄﾗｸﾄﾌﾟﾚｯｼｬｰ上下移動手動上昇BS
      MRD
      LD      B89  ; ﾌﾟﾚｯｼｬ 開端
      OR      M7092  ; D74=044ﾘﾄﾗｸﾄﾌﾟﾚｯｼｬｰ上昇
      ANB
      AND     X10A4  ; PS5 ｴｱ圧確認
      ANI     T200  ; ﾘﾄﾗｸﾄﾌﾟﾚｯｼｬ昇降上昇端遅延
      AND     M2417  ; ﾘﾄﾗｸﾄﾌﾟﾚｯｼｬｰ位置決め 後退端ﾌﾗｸﾞ
      OUT     M2500  ; ﾘﾄﾗｸﾄﾌﾟﾚｯｼｬｰ上下移動上昇IL
      MRD
      LDI     M30  ; 手動操作中
      OR      M2505  ; ﾘﾄﾗｸﾄﾌﾟﾚｯｼｬｰ上下移動手動上昇動作
      ANB
      LD      M15  ; 手動選択OK
      OR      L151  ; 試運転モード
      ANB
      AND     M2500  ; ﾘﾄﾗｸﾄﾌﾟﾚｯｼｬｰ上下移動上昇IL
      AND     X1005  ; 2PBL6 停止
      ANI     B4  ; 手動停止_TB
      ANI     M2515  ; ﾘﾄﾗｸﾄﾌﾟﾚｯｼｬｰ上下移動手動下降動作
      OUT     B0E6  ; ﾘﾄﾗｸﾄﾌﾟﾚｯｼｬ_上昇可TL
      MPP
      LDP     M2503  ; ﾘﾄﾗｸﾄﾌﾟﾚｯｼｬｰ上下移動手動上昇BS
      OR      M2505  ; ﾘﾄﾗｸﾄﾌﾟﾚｯｼｬｰ上下移動手動上昇動作
      AND     M2503  ; ﾘﾄﾗｸﾄﾌﾟﾚｯｼｬｰ上下移動手動上昇BS
      LD      M2505  ; ﾘﾄﾗｸﾄﾌﾟﾚｯｼｬｰ上下移動手動上昇動作
      ANI     L101  ; 寸動選択_TB
      ORB
      ANB
      AND     B0E6  ; ﾘﾄﾗｸﾄﾌﾟﾚｯｼｬ_上昇可TL
      OUT     M2505  ; ﾘﾄﾗｸﾄﾌﾟﾚｯｼｬｰ上下移動手動上昇動作
866   LD      SM400  ; 常時 ON
      MPS
      AND     B0E1  ; ﾘﾄﾗｸﾄﾌﾟﾚｯｼｬ_下降TB
      OUT     M2513  ; ﾘﾄﾗｸﾄﾌﾟﾚｯｼｬｰ上下移動手動下降BS
      MRD
      AND     X10A4  ; PS5 ｴｱ圧確認
      LD      B89  ; ﾌﾟﾚｯｼｬ 開端
      OR      M7090  ; D74=042ﾘﾄﾗｸﾄﾌﾟﾚｯｼｬｰ下降
      ANB
      ANI     T201  ; ﾘﾄﾗｸﾄﾌﾟﾚｯｼｬ昇降下降端遅延
      LD      T220  ; ﾘﾄﾗｸﾄﾌﾟﾚｯｼｬﾛｯｸ前進端遅延
      OR      B12A  ; ﾘﾄﾗｸﾄﾌﾟﾚｯｼｬ連結中
      OR      L151  ; 試運転モード
      ANB
      ANI     X108C  ; LS78 ﾘﾄﾗｸﾄﾌﾟﾚｯｼｬｰ前進端
      AND     M2417  ; ﾘﾄﾗｸﾄﾌﾟﾚｯｼｬｰ位置決め 後退端ﾌﾗｸﾞ
      OUT     M2510  ; ﾘﾄﾗｸﾄﾌﾟﾚｯｼｬｰ上下移動下降IL
      MRD
      LDI     M30  ; 手動操作中
      OR      M2515  ; ﾘﾄﾗｸﾄﾌﾟﾚｯｼｬｰ上下移動手動下降動作
      ANB
      LD      M15  ; 手動選択OK
      OR      L151  ; 試運転モード
      ANB
      AND     M2510  ; ﾘﾄﾗｸﾄﾌﾟﾚｯｼｬｰ上下移動下降IL
      AND     X1005  ; 2PBL6 停止
      ANI     B4  ; 手動停止_TB
      ANI     M2505  ; ﾘﾄﾗｸﾄﾌﾟﾚｯｼｬｰ上下移動手動上昇動作
      OUT     B0E7  ; ﾘﾄﾗｸﾄﾌﾟﾚｯｼｬ_下降可TL
      MPP
      LDP     M2513  ; ﾘﾄﾗｸﾄﾌﾟﾚｯｼｬｰ上下移動手動下降BS
      OR      M2515  ; ﾘﾄﾗｸﾄﾌﾟﾚｯｼｬｰ上下移動手動下降動作
      AND     M2513  ; ﾘﾄﾗｸﾄﾌﾟﾚｯｼｬｰ上下移動手動下降BS
      LD      M2515  ; ﾘﾄﾗｸﾄﾌﾟﾚｯｼｬｰ上下移動手動下降動作
      ANI     L101  ; 寸動選択_TB
      ORB
      ANB
      AND     B0E7  ; ﾘﾄﾗｸﾄﾌﾟﾚｯｼｬ_下降可TL
      OUT     M2515  ; ﾘﾄﾗｸﾄﾌﾟﾚｯｼｬｰ上下移動手動下降動作
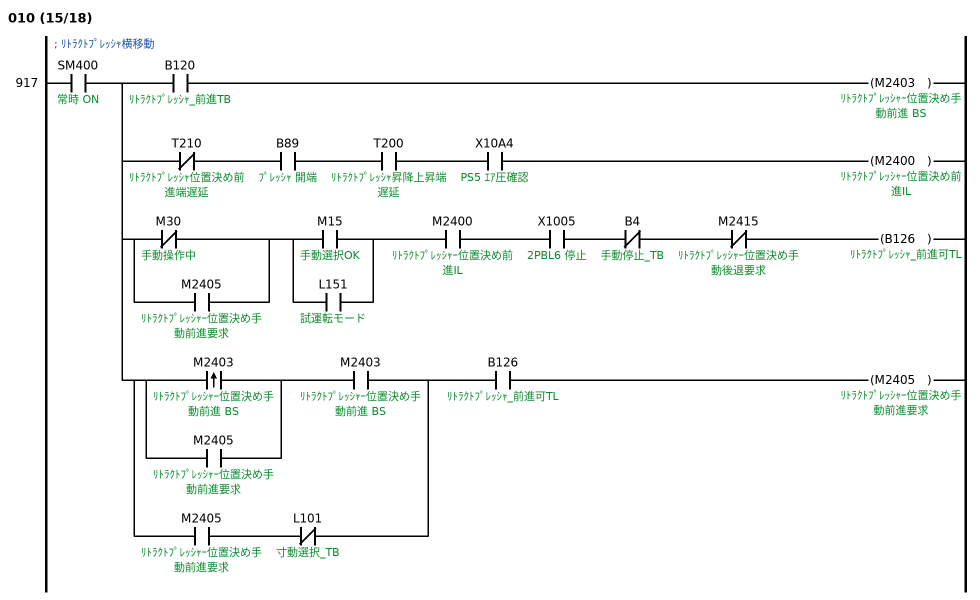
; ﾘﾄﾗｸﾄﾌﾟﾚｯｼｬ横移動
917   LD      SM400  ; 常時 ON
      MPS
      AND     B120  ; ﾘﾄﾗｸﾄﾌﾟﾚｯｼｬ_前進TB
      OUT     M2403  ; ﾘﾄﾗｸﾄﾌﾟﾚｯｼｬｰ位置決め手動前進 BS
      MRD
      ANI     T210  ; ﾘﾄﾗｸﾄﾌﾟﾚｯｼｬ位置決め前進端遅延
      AND     B89  ; ﾌﾟﾚｯｼｬ 開端
      AND     T200  ; ﾘﾄﾗｸﾄﾌﾟﾚｯｼｬ昇降上昇端遅延
      AND     X10A4  ; PS5 ｴｱ圧確認
      OUT     M2400  ; ﾘﾄﾗｸﾄﾌﾟﾚｯｼｬｰ位置決め前進IL
      MRD
      LDI     M30  ; 手動操作中
      OR      M2405  ; ﾘﾄﾗｸﾄﾌﾟﾚｯｼｬｰ位置決め手動前進要求
      ANB
      LD      M15  ; 手動選択OK
      OR      L151  ; 試運転モード
      ANB
      AND     M2400  ; ﾘﾄﾗｸﾄﾌﾟﾚｯｼｬｰ位置決め前進IL
      AND     X1005  ; 2PBL6 停止
      ANI     B4  ; 手動停止_TB
      ANI     M2415  ; ﾘﾄﾗｸﾄﾌﾟﾚｯｼｬｰ位置決め手動後退要求
      OUT     B126  ; ﾘﾄﾗｸﾄﾌﾟﾚｯｼｬ_前進可TL
      MPP
      LDP     M2403  ; ﾘﾄﾗｸﾄﾌﾟﾚｯｼｬｰ位置決め手動前進 BS
      OR      M2405  ; ﾘﾄﾗｸﾄﾌﾟﾚｯｼｬｰ位置決め手動前進要求
      AND     M2403  ; ﾘﾄﾗｸﾄﾌﾟﾚｯｼｬｰ位置決め手動前進 BS
      LD      M2405  ; ﾘﾄﾗｸﾄﾌﾟﾚｯｼｬｰ位置決め手動前進要求
      ANI     L101  ; 寸動選択_TB
      ORB
      ANB
      AND     B126  ; ﾘﾄﾗｸﾄﾌﾟﾚｯｼｬ_前進可TL
      OUT     M2405  ; ﾘﾄﾗｸﾄﾌﾟﾚｯｼｬｰ位置決め手動前進要求
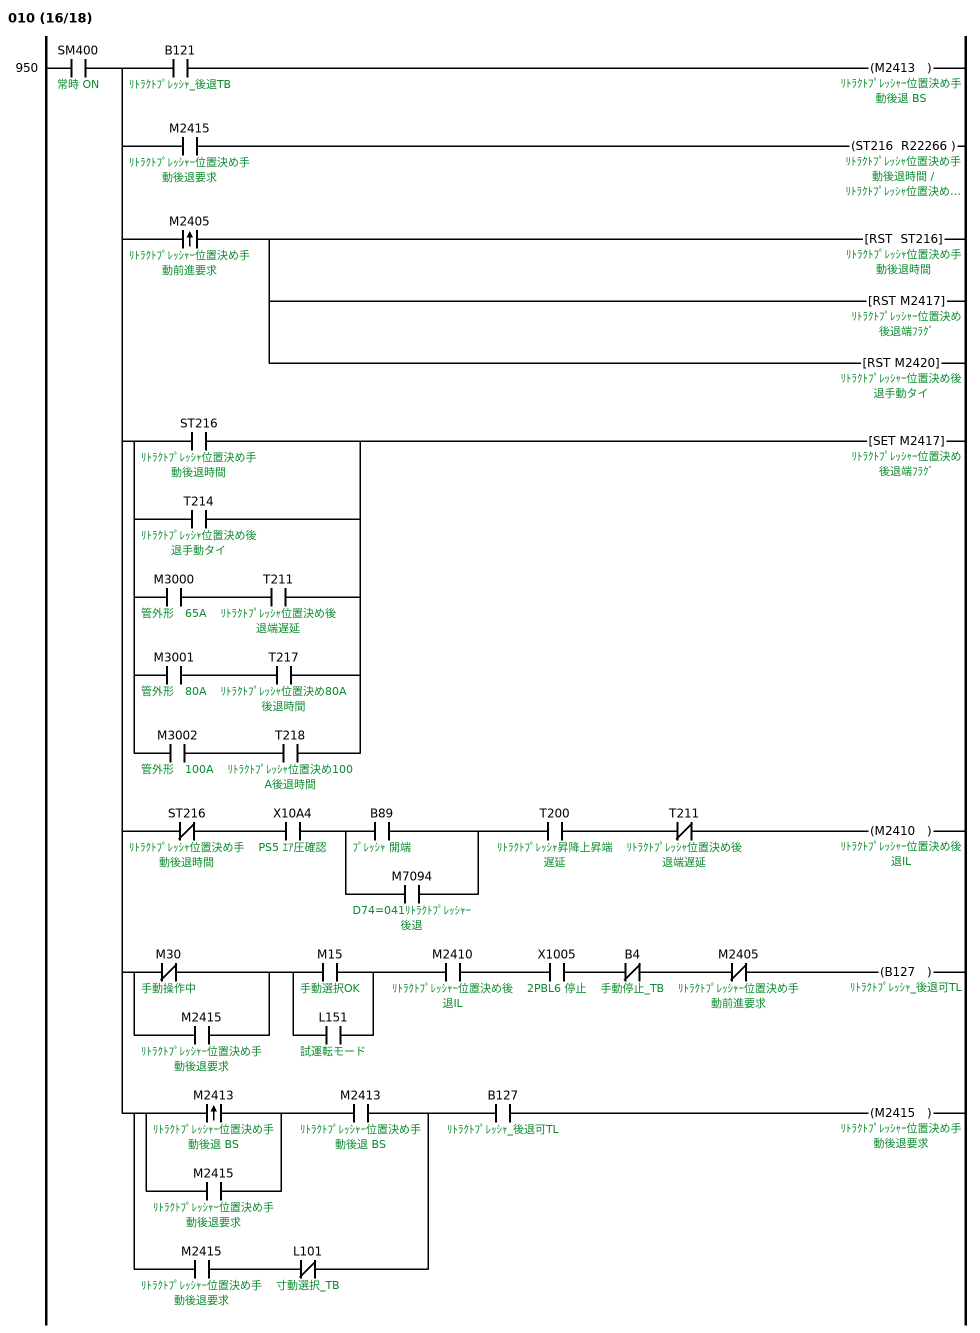
950   LD      SM400  ; 常時 ON
      MPS
      AND     B121  ; ﾘﾄﾗｸﾄﾌﾟﾚｯｼｬ_後退TB
      OUT     M2413  ; ﾘﾄﾗｸﾄﾌﾟﾚｯｼｬｰ位置決め手動後退 BS
      MRD
      AND     M2415  ; ﾘﾄﾗｸﾄﾌﾟﾚｯｼｬｰ位置決め手動後退要求
      OUT     ST216 R22266  ; ﾘﾄﾗｸﾄﾌﾟﾚｯｼｬ位置決め手動後退時間 / ﾘﾄﾗｸﾄﾌﾟﾚｯｼｬ位置決め手動時間
      MRD
      ANDP    M2405  ; ﾘﾄﾗｸﾄﾌﾟﾚｯｼｬｰ位置決め手動前進要求
      RST     ST216  ; ﾘﾄﾗｸﾄﾌﾟﾚｯｼｬ位置決め手動後退時間
      RST     M2417  ; ﾘﾄﾗｸﾄﾌﾟﾚｯｼｬｰ位置決め 後退端ﾌﾗｸﾞ
      RST     M2420  ; ﾘﾄﾗｸﾄﾌﾟﾚｯｼｬｰ位置決め後退手動タイ
      MRD
      LD      ST216  ; ﾘﾄﾗｸﾄﾌﾟﾚｯｼｬ位置決め手動後退時間
      OR      T214  ; ﾘﾄﾗｸﾄﾌﾟﾚｯｼｬ位置決め後退手動タイ
      LD      M3000  ; 管外形　65A
      AND     T211  ; ﾘﾄﾗｸﾄﾌﾟﾚｯｼｬ位置決め後退端遅延
      ORB
      LD      M3001  ; 管外形　80A
      AND     T217  ; ﾘﾄﾗｸﾄﾌﾟﾚｯｼｬ位置決め80A後退時間
      ORB
      LD      M3002  ; 管外形　100A
      AND     T218  ; ﾘﾄﾗｸﾄﾌﾟﾚｯｼｬ位置決め100A後退時間
      ORB
      ANB
      SET     M2417  ; ﾘﾄﾗｸﾄﾌﾟﾚｯｼｬｰ位置決め 後退端ﾌﾗｸﾞ
      MRD
      ANI     ST216  ; ﾘﾄﾗｸﾄﾌﾟﾚｯｼｬ位置決め手動後退時間
      AND     X10A4  ; PS5 ｴｱ圧確認
      LD      B89  ; ﾌﾟﾚｯｼｬ 開端
      OR      M7094  ; D74=041ﾘﾄﾗｸﾄﾌﾟﾚｯｼｬｰ後退
      ANB
      AND     T200  ; ﾘﾄﾗｸﾄﾌﾟﾚｯｼｬ昇降上昇端遅延
      ANI     T211  ; ﾘﾄﾗｸﾄﾌﾟﾚｯｼｬ位置決め後退端遅延
      OUT     M2410  ; ﾘﾄﾗｸﾄﾌﾟﾚｯｼｬｰ位置決め後退IL
      MRD
      LDI     M30  ; 手動操作中
      OR      M2415  ; ﾘﾄﾗｸﾄﾌﾟﾚｯｼｬｰ位置決め手動後退要求
      ANB
      LD      M15  ; 手動選択OK
      OR      L151  ; 試運転モード
      ANB
      AND     M2410  ; ﾘﾄﾗｸﾄﾌﾟﾚｯｼｬｰ位置決め後退IL
      AND     X1005  ; 2PBL6 停止
      ANI     B4  ; 手動停止_TB
      ANI     M2405  ; ﾘﾄﾗｸﾄﾌﾟﾚｯｼｬｰ位置決め手動前進要求
      OUT     B127  ; ﾘﾄﾗｸﾄﾌﾟﾚｯｼｬ_後退可TL
      MPP
      LDP     M2413  ; ﾘﾄﾗｸﾄﾌﾟﾚｯｼｬｰ位置決め手動後退 BS
      OR      M2415  ; ﾘﾄﾗｸﾄﾌﾟﾚｯｼｬｰ位置決め手動後退要求
      AND     M2413  ; ﾘﾄﾗｸﾄﾌﾟﾚｯｼｬｰ位置決め手動後退 BS
      LD      M2415  ; ﾘﾄﾗｸﾄﾌﾟﾚｯｼｬｰ位置決め手動後退要求
      ANI     L101  ; 寸動選択_TB
      ORB
      ANB
      AND     B127  ; ﾘﾄﾗｸﾄﾌﾟﾚｯｼｬ_後退可TL
      OUT     M2415  ; ﾘﾄﾗｸﾄﾌﾟﾚｯｼｬｰ位置決め手動後退要求
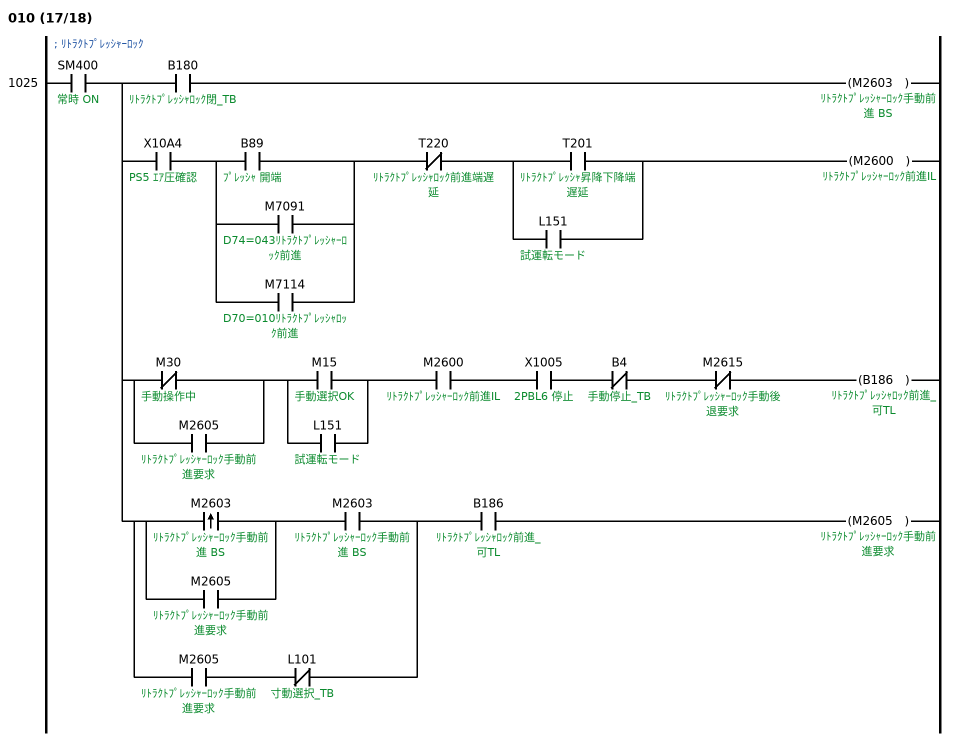
; ﾘﾄﾗｸﾄﾌﾟﾚｯｼｬｰﾛｯｸ
1025  LD      SM400  ; 常時 ON
      MPS
      AND     B180  ; ﾘﾄﾗｸﾄﾌﾟﾚｯｼｬﾛｯｸ閉_TB
      OUT     M2603  ; ﾘﾄﾗｸﾄﾌﾟﾚｯｼｬｰﾛｯｸ手動前進 BS
      MRD
      AND     X10A4  ; PS5 ｴｱ圧確認
      LD      B89  ; ﾌﾟﾚｯｼｬ 開端
      OR      M7091  ; D74=043ﾘﾄﾗｸﾄﾌﾟﾚｯｼｬｰﾛｯｸ前進
      OR      M7114  ; D70=010ﾘﾄﾗｸﾄﾌﾟﾚｯｼｬﾛｯｸ前進
      ANB
      ANI     T220  ; ﾘﾄﾗｸﾄﾌﾟﾚｯｼｬﾛｯｸ前進端遅延
      LD      T201  ; ﾘﾄﾗｸﾄﾌﾟﾚｯｼｬ昇降下降端遅延
      OR      L151  ; 試運転モード
      ANB
      OUT     M2600  ; ﾘﾄﾗｸﾄﾌﾟﾚｯｼｬｰﾛｯｸ前進IL
      MRD
      LDI     M30  ; 手動操作中
      OR      M2605  ; ﾘﾄﾗｸﾄﾌﾟﾚｯｼｬｰﾛｯｸ手動前進要求
      ANB
      LD      M15  ; 手動選択OK
      OR      L151  ; 試運転モード
      ANB
      AND     M2600  ; ﾘﾄﾗｸﾄﾌﾟﾚｯｼｬｰﾛｯｸ前進IL
      AND     X1005  ; 2PBL6 停止
      ANI     B4  ; 手動停止_TB
      ANI     M2615  ; ﾘﾄﾗｸﾄﾌﾟﾚｯｼｬｰﾛｯｸ手動後退要求
      OUT     B186  ; ﾘﾄﾗｸﾄﾌﾟﾚｯｼｬﾛｯｸ前進_可TL
      MPP
      LDP     M2603  ; ﾘﾄﾗｸﾄﾌﾟﾚｯｼｬｰﾛｯｸ手動前進 BS
      OR      M2605  ; ﾘﾄﾗｸﾄﾌﾟﾚｯｼｬｰﾛｯｸ手動前進要求
      AND     M2603  ; ﾘﾄﾗｸﾄﾌﾟﾚｯｼｬｰﾛｯｸ手動前進 BS
      LD      M2605  ; ﾘﾄﾗｸﾄﾌﾟﾚｯｼｬｰﾛｯｸ手動前進要求
      ANI     L101  ; 寸動選択_TB
      ORB
      ANB
      AND     B186  ; ﾘﾄﾗｸﾄﾌﾟﾚｯｼｬﾛｯｸ前進_可TL
      OUT     M2605  ; ﾘﾄﾗｸﾄﾌﾟﾚｯｼｬｰﾛｯｸ手動前進要求
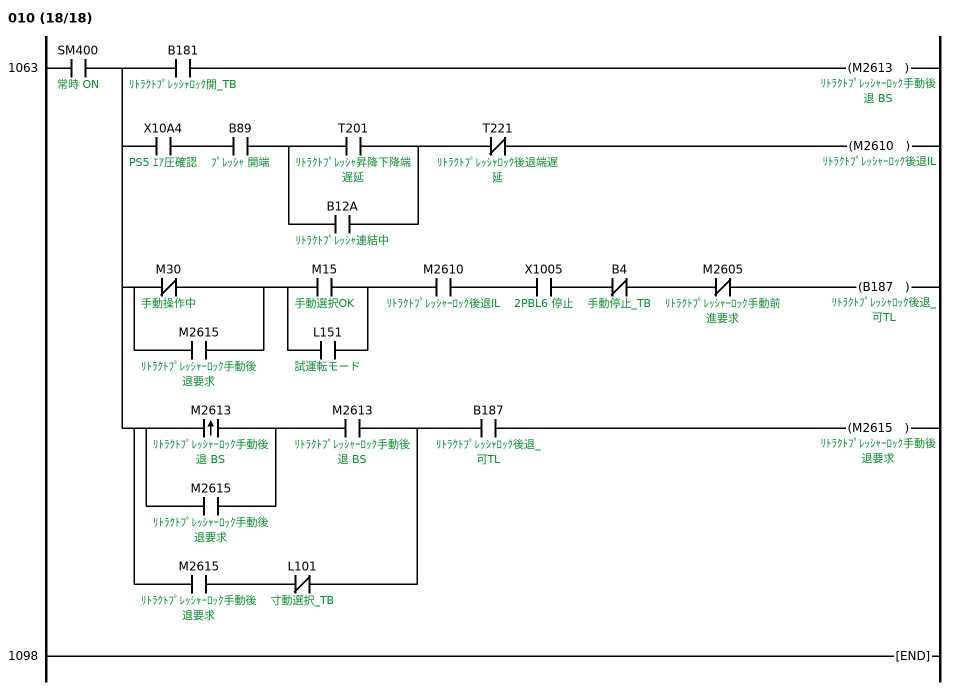
1063  LD      SM400  ; 常時 ON
      MPS
      AND     B181  ; ﾘﾄﾗｸﾄﾌﾟﾚｯｼｬﾛｯｸ開_TB
      OUT     M2613  ; ﾘﾄﾗｸﾄﾌﾟﾚｯｼｬｰﾛｯｸ手動後退 BS
      MRD
      AND     X10A4  ; PS5 ｴｱ圧確認
      AND     B89  ; ﾌﾟﾚｯｼｬ 開端
      LD      T201  ; ﾘﾄﾗｸﾄﾌﾟﾚｯｼｬ昇降下降端遅延
      OR      B12A  ; ﾘﾄﾗｸﾄﾌﾟﾚｯｼｬ連結中
      ANB
      ANI     T221  ; ﾘﾄﾗｸﾄﾌﾟﾚｯｼｬﾛｯｸ後退端遅延
      OUT     M2610  ; ﾘﾄﾗｸﾄﾌﾟﾚｯｼｬｰﾛｯｸ後退IL
      MRD
      LDI     M30  ; 手動操作中
      OR      M2615  ; ﾘﾄﾗｸﾄﾌﾟﾚｯｼｬｰﾛｯｸ手動後退要求
      ANB
      LD      M15  ; 手動選択OK
      OR      L151  ; 試運転モード
      ANB
      AND     M2610  ; ﾘﾄﾗｸﾄﾌﾟﾚｯｼｬｰﾛｯｸ後退IL
      AND     X1005  ; 2PBL6 停止
      ANI     B4  ; 手動停止_TB
      ANI     M2605  ; ﾘﾄﾗｸﾄﾌﾟﾚｯｼｬｰﾛｯｸ手動前進要求
      OUT     B187  ; ﾘﾄﾗｸﾄﾌﾟﾚｯｼｬﾛｯｸ後退_可TL
      MPP
      LDP     M2613  ; ﾘﾄﾗｸﾄﾌﾟﾚｯｼｬｰﾛｯｸ手動後退 BS
      OR      M2615  ; ﾘﾄﾗｸﾄﾌﾟﾚｯｼｬｰﾛｯｸ手動後退要求
      AND     M2613  ; ﾘﾄﾗｸﾄﾌﾟﾚｯｼｬｰﾛｯｸ手動後退 BS
      LD      M2615  ; ﾘﾄﾗｸﾄﾌﾟﾚｯｼｬｰﾛｯｸ手動後退要求
      ANI     L101  ; 寸動選択_TB
      ORB
      ANB
      AND     B187  ; ﾘﾄﾗｸﾄﾌﾟﾚｯｼｬﾛｯｸ後退_可TL
      OUT     M2615  ; ﾘﾄﾗｸﾄﾌﾟﾚｯｼｬｰﾛｯｸ手動後退要求
1098  END
END_PROGRAM

PROGRAM 011  // 手動段取替え
; 
      P1100
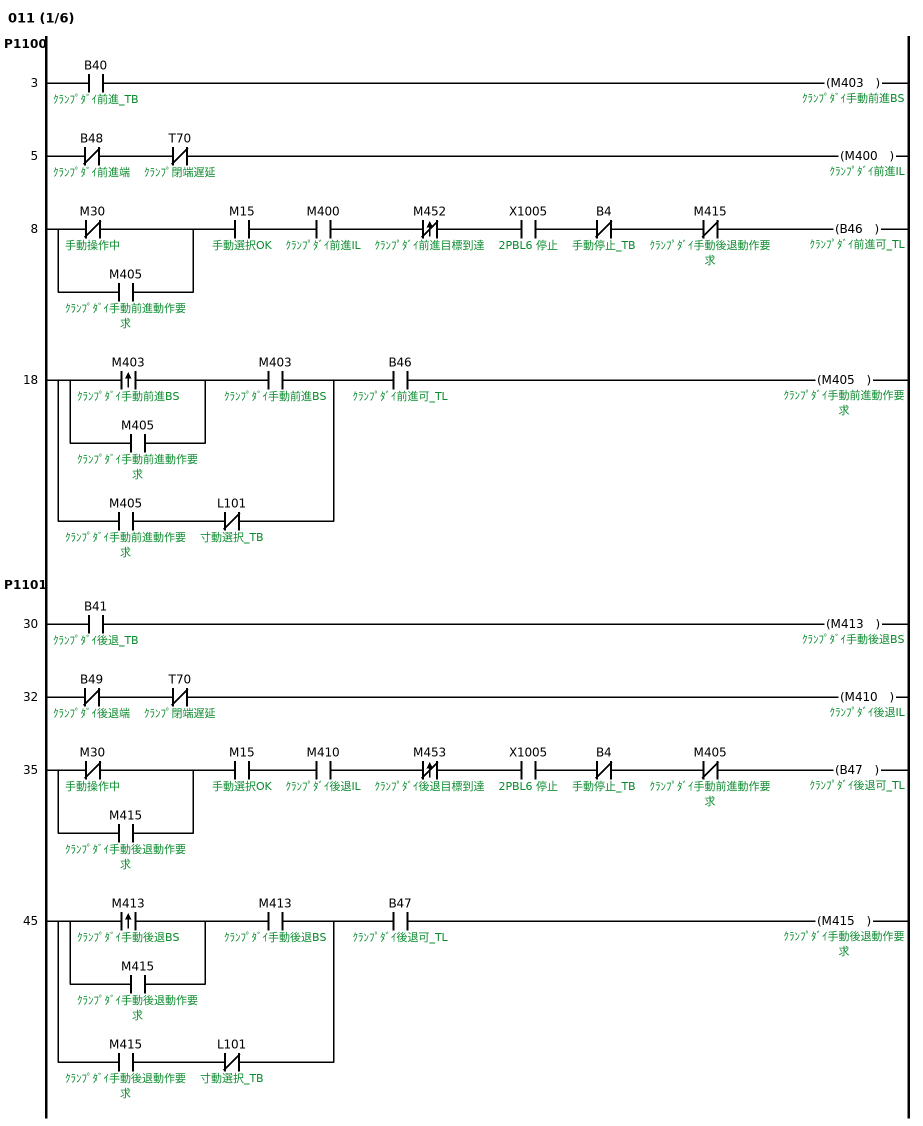
3     LD      B40  ; ｸﾗﾝﾌﾟﾀﾞｲ前進_TB
      OUT     M403  ; ｸﾗﾝﾌﾟﾀﾞｲ手動前進BS
5     LDI     B48  ; ｸﾗﾝﾌﾟﾀﾞｲ前進端
      ANI     T70  ; ｸﾗﾝﾌﾟ閉端遅延
      OUT     M400  ; ｸﾗﾝﾌﾟﾀﾞｲ前進IL
8     LDI     M30  ; 手動操作中
      OR      M405  ; ｸﾗﾝﾌﾟﾀﾞｲ手動前進動作要求
      AND     M15  ; 手動選択OK
      AND     M400  ; ｸﾗﾝﾌﾟﾀﾞｲ前進IL
      ANDPI   M452  ; ｸﾗﾝﾌﾟﾀﾞｲ前進目標到達
      AND     X1005  ; 2PBL6 停止
      ANI     B4  ; 手動停止_TB
      ANI     M415  ; ｸﾗﾝﾌﾟﾀﾞｲ手動後退動作要求
      OUT     B46  ; ｸﾗﾝﾌﾟﾀﾞｲ前進可_TL
18    LDP     M403  ; ｸﾗﾝﾌﾟﾀﾞｲ手動前進BS
      OR      M405  ; ｸﾗﾝﾌﾟﾀﾞｲ手動前進動作要求
      AND     M403  ; ｸﾗﾝﾌﾟﾀﾞｲ手動前進BS
      LD      M405  ; ｸﾗﾝﾌﾟﾀﾞｲ手動前進動作要求
      ANI     L101  ; 寸動選択_TB
      ORB
      AND     B46  ; ｸﾗﾝﾌﾟﾀﾞｲ前進可_TL
      OUT     M405  ; ｸﾗﾝﾌﾟﾀﾞｲ手動前進動作要求
; 
      P1101
30    LD      B41  ; ｸﾗﾝﾌﾟﾀﾞｲ後退_TB
      OUT     M413  ; ｸﾗﾝﾌﾟﾀﾞｲ手動後退BS
32    LDI     B49  ; ｸﾗﾝﾌﾟﾀﾞｲ後退端
      ANI     T70  ; ｸﾗﾝﾌﾟ閉端遅延
      OUT     M410  ; ｸﾗﾝﾌﾟﾀﾞｲ後退IL
35    LDI     M30  ; 手動操作中
      OR      M415  ; ｸﾗﾝﾌﾟﾀﾞｲ手動後退動作要求
      AND     M15  ; 手動選択OK
      AND     M410  ; ｸﾗﾝﾌﾟﾀﾞｲ後退IL
      ANDPI   M453  ; ｸﾗﾝﾌﾟﾀﾞｲ後退目標到達
      AND     X1005  ; 2PBL6 停止
      ANI     B4  ; 手動停止_TB
      ANI     M405  ; ｸﾗﾝﾌﾟﾀﾞｲ手動前進動作要求
      OUT     B47  ; ｸﾗﾝﾌﾟﾀﾞｲ後退可_TL
45    LDP     M413  ; ｸﾗﾝﾌﾟﾀﾞｲ手動後退BS
      OR      M415  ; ｸﾗﾝﾌﾟﾀﾞｲ手動後退動作要求
      AND     M413  ; ｸﾗﾝﾌﾟﾀﾞｲ手動後退BS
      LD      M415  ; ｸﾗﾝﾌﾟﾀﾞｲ手動後退動作要求
      ANI     L101  ; 寸動選択_TB
      ORB
      AND     B47  ; ｸﾗﾝﾌﾟﾀﾞｲ後退可_TL
      OUT     M415  ; ｸﾗﾝﾌﾟﾀﾞｲ手動後退動作要求
      P1102
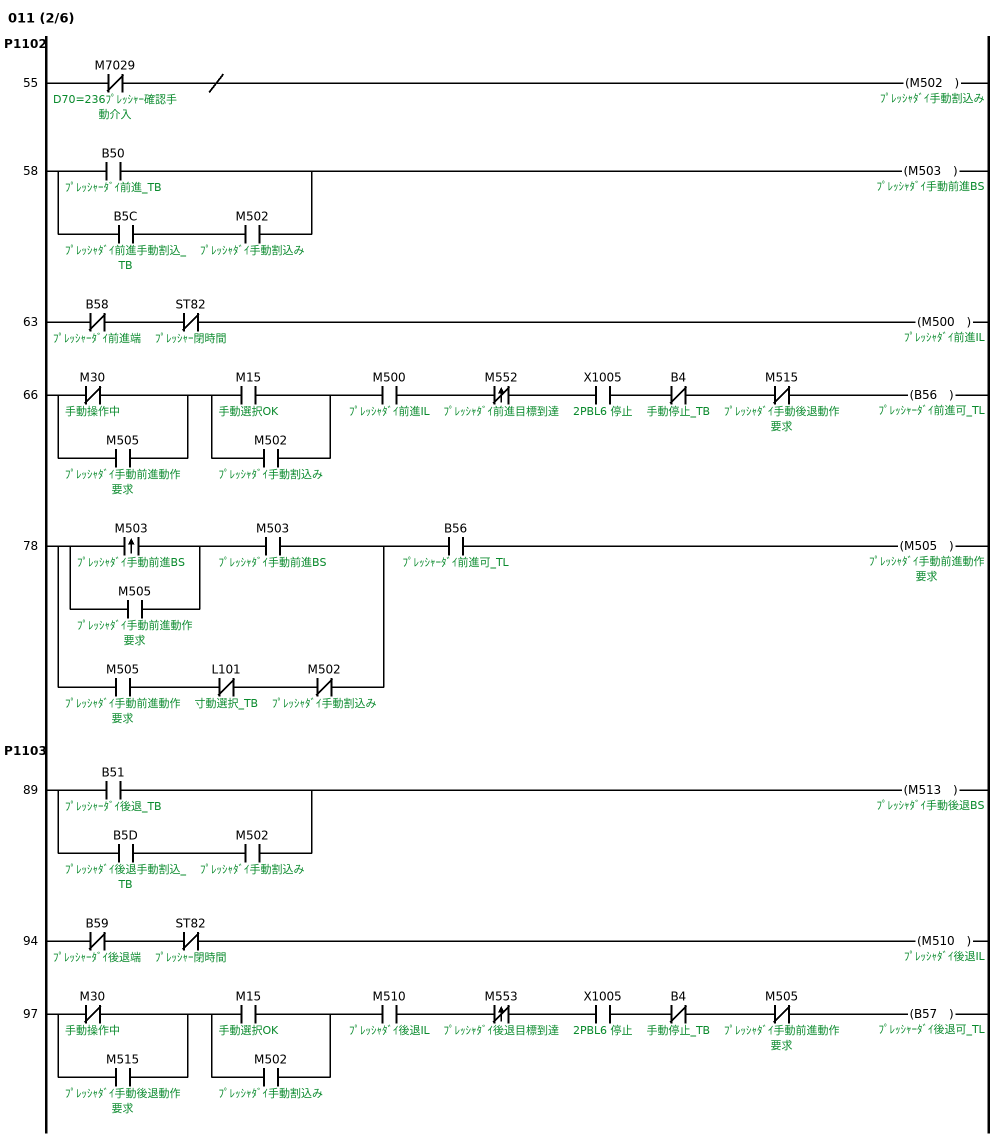
55    LDI     M7029  ; D70=236ﾌﾟﾚｯｼｬｰ確認手動介入
      INV
      OUT     M502  ; ﾌﾟﾚｯｼｬﾀﾞｲ手動割込み
58    LD      B50  ; ﾌﾟﾚｯｼｬｰﾀﾞｲ前進_TB
      LD      B5C  ; ﾌﾟﾚｯｼｬﾀﾞｲ前進手動割込_TB
      AND     M502  ; ﾌﾟﾚｯｼｬﾀﾞｲ手動割込み
      ORB
      OUT     M503  ; ﾌﾟﾚｯｼｬﾀﾞｲ手動前進BS
63    LDI     B58  ; ﾌﾟﾚｯｼｬｰﾀﾞｲ前進端
      ANI     ST82  ; ﾌﾟﾚｯｼｬｰ閉時間
      OUT     M500  ; ﾌﾟﾚｯｼｬﾀﾞｲ前進IL
66    LDI     M30  ; 手動操作中
      OR      M505  ; ﾌﾟﾚｯｼｬﾀﾞｲ手動前進動作要求
      LD      M15  ; 手動選択OK
      OR      M502  ; ﾌﾟﾚｯｼｬﾀﾞｲ手動割込み
      ANB
      AND     M500  ; ﾌﾟﾚｯｼｬﾀﾞｲ前進IL
      ANDPI   M552  ; ﾌﾟﾚｯｼｬﾀﾞｲ前進目標到達
      AND     X1005  ; 2PBL6 停止
      ANI     B4  ; 手動停止_TB
      ANI     M515  ; ﾌﾟﾚｯｼｬﾀﾞｲ手動後退動作要求
      OUT     B56  ; ﾌﾟﾚｯｼｬｰﾀﾞｲ前進可_TL
78    LDP     M503  ; ﾌﾟﾚｯｼｬﾀﾞｲ手動前進BS
      OR      M505  ; ﾌﾟﾚｯｼｬﾀﾞｲ手動前進動作要求
      AND     M503  ; ﾌﾟﾚｯｼｬﾀﾞｲ手動前進BS
      LD      M505  ; ﾌﾟﾚｯｼｬﾀﾞｲ手動前進動作要求
      ANI     L101  ; 寸動選択_TB
      ANI     M502  ; ﾌﾟﾚｯｼｬﾀﾞｲ手動割込み
      ORB
      AND     B56  ; ﾌﾟﾚｯｼｬｰﾀﾞｲ前進可_TL
      OUT     M505  ; ﾌﾟﾚｯｼｬﾀﾞｲ手動前進動作要求
      P1103
89    LD      B51  ; ﾌﾟﾚｯｼｬｰﾀﾞｲ後退_TB
      LD      B5D  ; ﾌﾟﾚｯｼｬﾀﾞｲ後退手動割込_TB
      AND     M502  ; ﾌﾟﾚｯｼｬﾀﾞｲ手動割込み
      ORB
      OUT     M513  ; ﾌﾟﾚｯｼｬﾀﾞｲ手動後退BS
94    LDI     B59  ; ﾌﾟﾚｯｼｬｰﾀﾞｲ後退端
      ANI     ST82  ; ﾌﾟﾚｯｼｬｰ閉時間
      OUT     M510  ; ﾌﾟﾚｯｼｬﾀﾞｲ後退IL
97    LDI     M30  ; 手動操作中
      OR      M515  ; ﾌﾟﾚｯｼｬﾀﾞｲ手動後退動作要求
      LD      M15  ; 手動選択OK
      OR      M502  ; ﾌﾟﾚｯｼｬﾀﾞｲ手動割込み
      ANB
      AND     M510  ; ﾌﾟﾚｯｼｬﾀﾞｲ後退IL
      ANDPI   M553  ; ﾌﾟﾚｯｼｬﾀﾞｲ後退目標到達
      AND     X1005  ; 2PBL6 停止
      ANI     B4  ; 手動停止_TB
      ANI     M505  ; ﾌﾟﾚｯｼｬﾀﾞｲ手動前進動作要求
      OUT     B57  ; ﾌﾟﾚｯｼｬｰﾀﾞｲ後退可_TL
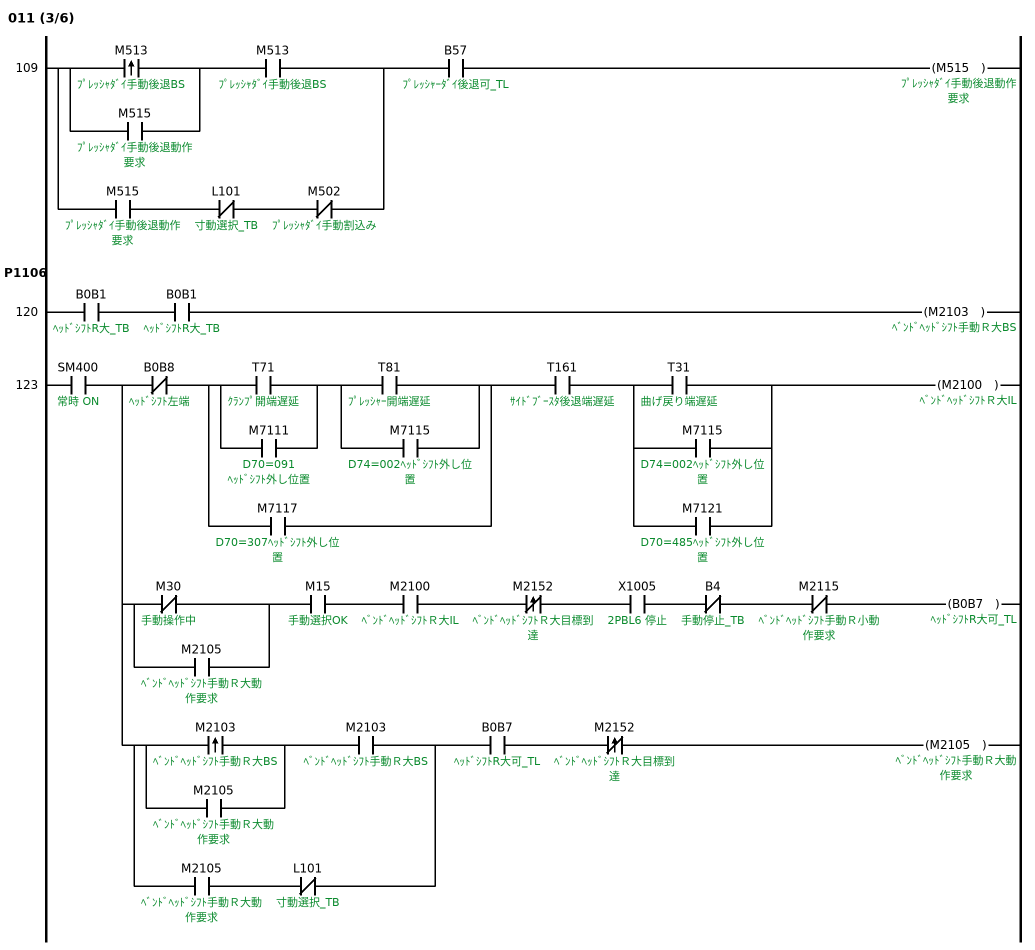
109   LDP     M513  ; ﾌﾟﾚｯｼｬﾀﾞｲ手動後退BS
      OR      M515  ; ﾌﾟﾚｯｼｬﾀﾞｲ手動後退動作要求
      AND     M513  ; ﾌﾟﾚｯｼｬﾀﾞｲ手動後退BS
      LD      M515  ; ﾌﾟﾚｯｼｬﾀﾞｲ手動後退動作要求
      ANI     L101  ; 寸動選択_TB
      ANI     M502  ; ﾌﾟﾚｯｼｬﾀﾞｲ手動割込み
      ORB
      AND     B57  ; ﾌﾟﾚｯｼｬｰﾀﾞｲ後退可_TL
      OUT     M515  ; ﾌﾟﾚｯｼｬﾀﾞｲ手動後退動作要求
      P1106
120   LD      B0B1  ; ﾍｯﾄﾞｼﾌﾄR大_TB
      AND     B0B1  ; ﾍｯﾄﾞｼﾌﾄR大_TB
      OUT     M2103  ; ﾍﾞﾝﾄﾞﾍｯﾄﾞｼﾌﾄ手動Ｒ大BS
123   LD      SM400  ; 常時 ON
      MPS
      ANI     B0B8  ; ﾍｯﾄﾞｼﾌﾄ左端
      LD      T71  ; ｸﾗﾝﾌﾟ開端遅延
      OR      M7111  ; D70=091 ﾍｯﾄﾞｼﾌﾄ外し位置
      LD      T81  ; ﾌﾟﾚｯｼｬｰ開端遅延
      OR      M7115  ; D74=002ﾍｯﾄﾞｼﾌﾄ外し位置
      ANB
      OR      M7117  ; D70=307ﾍｯﾄﾞｼﾌﾄ外し位置
      ANB
      AND     T161  ; ｻｲﾄﾞﾌﾞｰｽﾀ後退端遅延
      LD      T31  ; 曲げ戻り端遅延
      OR      M7115  ; D74=002ﾍｯﾄﾞｼﾌﾄ外し位置
      OR      M7121  ; D70=485ﾍｯﾄﾞｼﾌﾄ外し位置
      ANB
      OUT     M2100  ; ﾍﾞﾝﾄﾞﾍｯﾄﾞｼﾌﾄＲ大IL
      MRD
      LDI     M30  ; 手動操作中
      OR      M2105  ; ﾍﾞﾝﾄﾞﾍｯﾄﾞｼﾌﾄ手動Ｒ大動作要求
      ANB
      AND     M15  ; 手動選択OK
      AND     M2100  ; ﾍﾞﾝﾄﾞﾍｯﾄﾞｼﾌﾄＲ大IL
      ANDPI   M2152  ; ﾍﾞﾝﾄﾞﾍｯﾄﾞｼﾌﾄＲ大目標到達
      AND     X1005  ; 2PBL6 停止
      ANI     B4  ; 手動停止_TB
      ANI     M2115  ; ﾍﾞﾝﾄﾞﾍｯﾄﾞｼﾌﾄ手動Ｒ小動作要求
      OUT     B0B7  ; ﾍｯﾄﾞｼﾌﾄR大可_TL
      MPP
      LDP     M2103  ; ﾍﾞﾝﾄﾞﾍｯﾄﾞｼﾌﾄ手動Ｒ大BS
      OR      M2105  ; ﾍﾞﾝﾄﾞﾍｯﾄﾞｼﾌﾄ手動Ｒ大動作要求
      AND     M2103  ; ﾍﾞﾝﾄﾞﾍｯﾄﾞｼﾌﾄ手動Ｒ大BS
      LD      M2105  ; ﾍﾞﾝﾄﾞﾍｯﾄﾞｼﾌﾄ手動Ｒ大動作要求
      ANI     L101  ; 寸動選択_TB
      ORB
      ANB
      AND     B0B7  ; ﾍｯﾄﾞｼﾌﾄR大可_TL
      ANDPI   M2152  ; ﾍﾞﾝﾄﾞﾍｯﾄﾞｼﾌﾄＲ大目標到達
      OUT     M2105  ; ﾍﾞﾝﾄﾞﾍｯﾄﾞｼﾌﾄ手動Ｒ大動作要求
      P1107
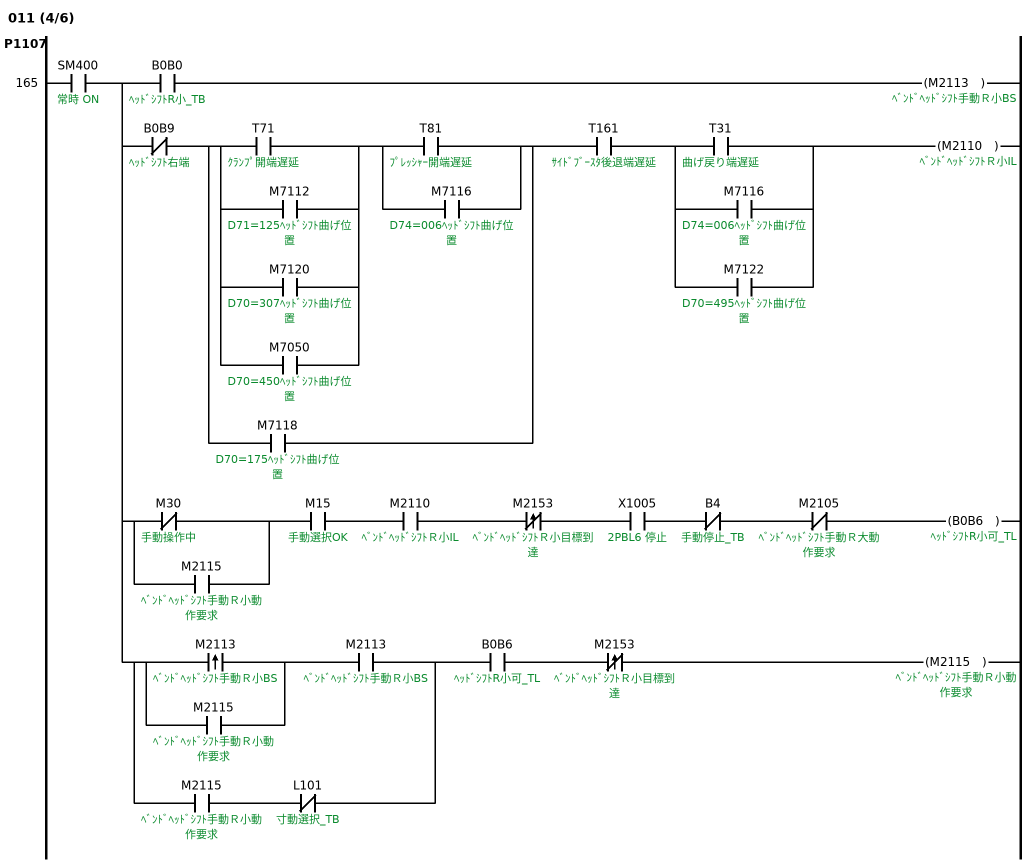
165   LD      SM400  ; 常時 ON
      MPS
      AND     B0B0  ; ﾍｯﾄﾞｼﾌﾄR小_TB
      OUT     M2113  ; ﾍﾞﾝﾄﾞﾍｯﾄﾞｼﾌﾄ手動Ｒ小BS
      MRD
      ANI     B0B9  ; ﾍｯﾄﾞｼﾌﾄ右端
      LD      T71  ; ｸﾗﾝﾌﾟ開端遅延
      OR      M7112  ; D71=125ﾍｯﾄﾞｼﾌﾄ曲げ位置
      OR      M7120  ; D70=307ﾍｯﾄﾞｼﾌﾄ曲げ位置
      OR      M7050  ; D70=450ﾍｯﾄﾞｼﾌﾄ曲げ位置
      LD      T81  ; ﾌﾟﾚｯｼｬｰ開端遅延
      OR      M7116  ; D74=006ﾍｯﾄﾞｼﾌﾄ曲げ位置
      ANB
      OR      M7118  ; D70=175ﾍｯﾄﾞｼﾌﾄ曲げ位置
      ANB
      AND     T161  ; ｻｲﾄﾞﾌﾞｰｽﾀ後退端遅延
      LD      T31  ; 曲げ戻り端遅延
      OR      M7116  ; D74=006ﾍｯﾄﾞｼﾌﾄ曲げ位置
      OR      M7122  ; D70=495ﾍｯﾄﾞｼﾌﾄ曲げ位置
      ANB
      OUT     M2110  ; ﾍﾞﾝﾄﾞﾍｯﾄﾞｼﾌﾄＲ小IL
      MRD
      LDI     M30  ; 手動操作中
      OR      M2115  ; ﾍﾞﾝﾄﾞﾍｯﾄﾞｼﾌﾄ手動Ｒ小動作要求
      ANB
      AND     M15  ; 手動選択OK
      AND     M2110  ; ﾍﾞﾝﾄﾞﾍｯﾄﾞｼﾌﾄＲ小IL
      ANDPI   M2153  ; ﾍﾞﾝﾄﾞﾍｯﾄﾞｼﾌﾄＲ小目標到達
      AND     X1005  ; 2PBL6 停止
      ANI     B4  ; 手動停止_TB
      ANI     M2105  ; ﾍﾞﾝﾄﾞﾍｯﾄﾞｼﾌﾄ手動Ｒ大動作要求
      OUT     B0B6  ; ﾍｯﾄﾞｼﾌﾄR小可_TL
      MPP
      LDP     M2113  ; ﾍﾞﾝﾄﾞﾍｯﾄﾞｼﾌﾄ手動Ｒ小BS
      OR      M2115  ; ﾍﾞﾝﾄﾞﾍｯﾄﾞｼﾌﾄ手動Ｒ小動作要求
      AND     M2113  ; ﾍﾞﾝﾄﾞﾍｯﾄﾞｼﾌﾄ手動Ｒ小BS
      LD      M2115  ; ﾍﾞﾝﾄﾞﾍｯﾄﾞｼﾌﾄ手動Ｒ小動作要求
      ANI     L101  ; 寸動選択_TB
      ORB
      ANB
      AND     B0B6  ; ﾍｯﾄﾞｼﾌﾄR小可_TL
      ANDPI   M2153  ; ﾍﾞﾝﾄﾞﾍｯﾄﾞｼﾌﾄＲ小目標到達
      OUT     M2115  ; ﾍﾞﾝﾄﾞﾍｯﾄﾞｼﾌﾄ手動Ｒ小動作要求
      P1108
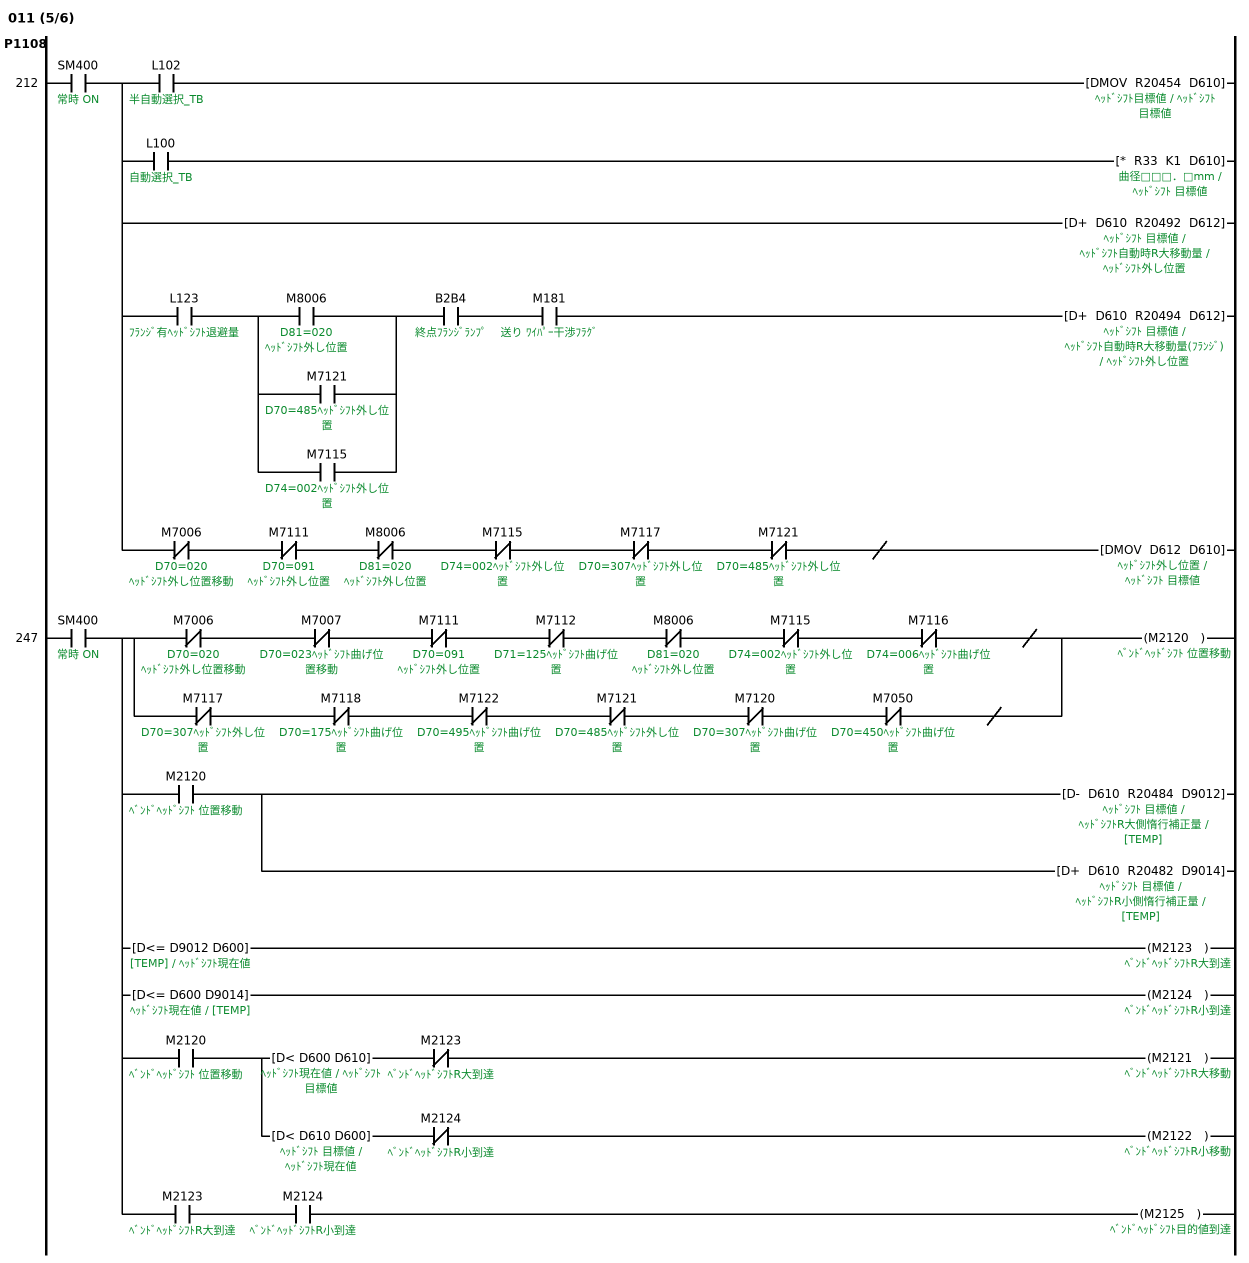
212   LD      SM400  ; 常時 ON
      MPS
      AND     L102  ; 半自動選択_TB
      DMOV    R20454 D610  ; ﾍｯﾄﾞｼﾌﾄ目標値 / ﾍｯﾄﾞｼﾌﾄ 目標値
      MRD
      AND     L100  ; 自動選択_TB
      *       R33 K1 D610  ; 曲径□□□．□mm
      MPP
      D+      D610 R20492 D612  ; ﾍｯﾄﾞｼﾌﾄ自動時R大移動量 / ﾍｯﾄﾞｼﾌﾄ外し位置
      MPS
      AND     L123  ; ﾌﾗﾝｼﾞ有ﾍｯﾄﾞｼﾌﾄ退避量
      LD      M8006  ; D81=020 ﾍｯﾄﾞｼﾌﾄ外し位置
      OR      M7121  ; D70=485ﾍｯﾄﾞｼﾌﾄ外し位置
      OR      M7115  ; D74=002ﾍｯﾄﾞｼﾌﾄ外し位置
      ANB
      AND     B2B4  ; 終点ﾌﾗﾝｼﾞﾗﾝﾌﾟ
      AND     M181  ; 送り ﾜｲﾊﾟｰ干渉ﾌﾗｸﾞ
      D+      D610 R20494 D612  ; ﾍｯﾄﾞｼﾌﾄ自動時R大移動量(ﾌﾗﾝｼﾞ)
      MPP
      ANI     M7006  ; D70=020 ﾍｯﾄﾞｼﾌﾄ外し位置移動
      ANI     M7111  ; D70=091 ﾍｯﾄﾞｼﾌﾄ外し位置
      ANI     M8006  ; D81=020 ﾍｯﾄﾞｼﾌﾄ外し位置
      ANI     M7115  ; D74=002ﾍｯﾄﾞｼﾌﾄ外し位置
      ANI     M7117  ; D70=307ﾍｯﾄﾞｼﾌﾄ外し位置
      ANI     M7121  ; D70=485ﾍｯﾄﾞｼﾌﾄ外し位置
      INV
      DMOV    D612 D610
247   LD      SM400  ; 常時 ON
      MPS
      LDI     M7006  ; D70=020 ﾍｯﾄﾞｼﾌﾄ外し位置移動
      ANI     M7007  ; D70=023ﾍｯﾄﾞｼﾌﾄ曲げ位置移動
      ANI     M7111  ; D70=091 ﾍｯﾄﾞｼﾌﾄ外し位置
      ANI     M7112  ; D71=125ﾍｯﾄﾞｼﾌﾄ曲げ位置
      ANI     M8006  ; D81=020 ﾍｯﾄﾞｼﾌﾄ外し位置
      ANI     M7115  ; D74=002ﾍｯﾄﾞｼﾌﾄ外し位置
      ANI     M7116  ; D74=006ﾍｯﾄﾞｼﾌﾄ曲げ位置
      INV
      LDI     M7117  ; D70=307ﾍｯﾄﾞｼﾌﾄ外し位置
      ANI     M7118  ; D70=175ﾍｯﾄﾞｼﾌﾄ曲げ位置
      ANI     M7122  ; D70=495ﾍｯﾄﾞｼﾌﾄ曲げ位置
      ANI     M7121  ; D70=485ﾍｯﾄﾞｼﾌﾄ外し位置
      ANI     M7120  ; D70=307ﾍｯﾄﾞｼﾌﾄ曲げ位置
      ANI     M7050  ; D70=450ﾍｯﾄﾞｼﾌﾄ曲げ位置
      INV
      ORB
      ANB
      OUT     M2120  ; ﾍﾞﾝﾄﾞﾍｯﾄﾞｼﾌﾄ 位置移動
      MRD
      AND     M2120  ; ﾍﾞﾝﾄﾞﾍｯﾄﾞｼﾌﾄ 位置移動
      D-      D610 R20484 D9012  ; ﾍｯﾄﾞｼﾌﾄR大側惰行補正量 / [TEMP]
      D+      D610 R20482 D9014  ; ﾍｯﾄﾞｼﾌﾄR小側惰行補正量 / [TEMP]
      MRD
      ANDD<=  D9012 D600  ; [TEMP] / ﾍｯﾄﾞｼﾌﾄ現在値
      OUT     M2123  ; ﾍﾞﾝﾄﾞﾍｯﾄﾞｼﾌﾄR大到達
      MRD
      ANDD<=  D600 D9014  ; ﾍｯﾄﾞｼﾌﾄ現在値 / [TEMP]
      OUT     M2124  ; ﾍﾞﾝﾄﾞﾍｯﾄﾞｼﾌﾄR小到達
      MRD
      AND     M2120  ; ﾍﾞﾝﾄﾞﾍｯﾄﾞｼﾌﾄ 位置移動
      MPS
      ANDD<   D600 D610  ; ﾍｯﾄﾞｼﾌﾄ現在値 / ﾍｯﾄﾞｼﾌﾄ 目標値
      ANI     M2123  ; ﾍﾞﾝﾄﾞﾍｯﾄﾞｼﾌﾄR大到達
      OUT     M2121  ; ﾍﾞﾝﾄﾞﾍｯﾄﾞｼﾌﾄR大移動
      MPP
      ANDD<   D610 D600  ; ﾍｯﾄﾞｼﾌﾄ 目標値 / ﾍｯﾄﾞｼﾌﾄ現在値
      ANI     M2124  ; ﾍﾞﾝﾄﾞﾍｯﾄﾞｼﾌﾄR小到達
      OUT     M2122  ; ﾍﾞﾝﾄﾞﾍｯﾄﾞｼﾌﾄR小移動
      MPP
      AND     M2123  ; ﾍﾞﾝﾄﾞﾍｯﾄﾞｼﾌﾄR大到達
      AND     M2124  ; ﾍﾞﾝﾄﾞﾍｯﾄﾞｼﾌﾄR小到達
      OUT     M2125  ; ﾍﾞﾝﾄﾞﾍｯﾄﾞｼﾌﾄ目的値到達
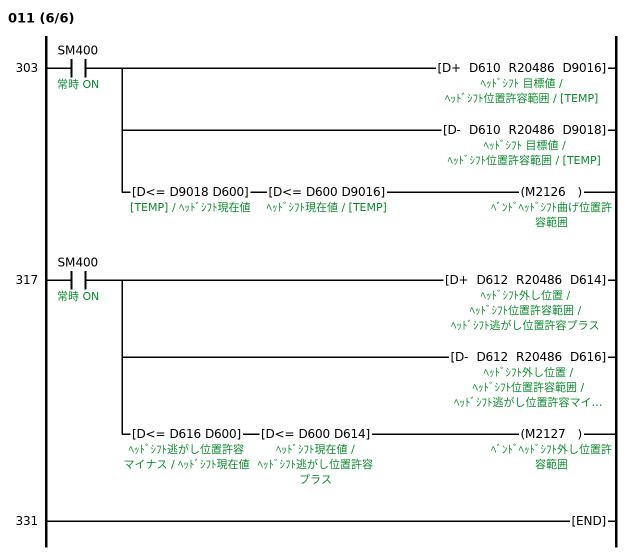
303   LD      SM400  ; 常時 ON
      D+      D610 R20486 D9016  ; ﾍｯﾄﾞｼﾌﾄ位置許容範囲 / [TEMP]
      D-      D610 R20486 D9018  ; [TEMP]
      ANDD<=  D9018 D600  ; [TEMP] / ﾍｯﾄﾞｼﾌﾄ現在値
      ANDD<=  D600 D9016  ; ﾍｯﾄﾞｼﾌﾄ現在値 / [TEMP]
      OUT     M2126  ; ﾍﾞﾝﾄﾞﾍｯﾄﾞｼﾌﾄ曲げ位置許容範囲
317   LD      SM400  ; 常時 ON
      D+      D612 R20486 D614  ; ﾍｯﾄﾞｼﾌﾄ逃がし位置許容プラス
      D-      D612 R20486 D616  ; ﾍｯﾄﾞｼﾌﾄ逃がし位置許容マイナス
      ANDD<=  D616 D600  ; ﾍｯﾄﾞｼﾌﾄ逃がし位置許容マイナス / ﾍｯﾄﾞｼﾌﾄ現在値
      ANDD<=  D600 D614  ; ﾍｯﾄﾞｼﾌﾄ現在値 / ﾍｯﾄﾞｼﾌﾄ逃がし位置許容プラス
      OUT     M2127  ; ﾍﾞﾝﾄﾞﾍｯﾄﾞｼﾌﾄ外し位置許容範囲
331   END
END_PROGRAM

PROGRAM 012  // 手動ｻﾌﾞ自動開始
; 
      P1201
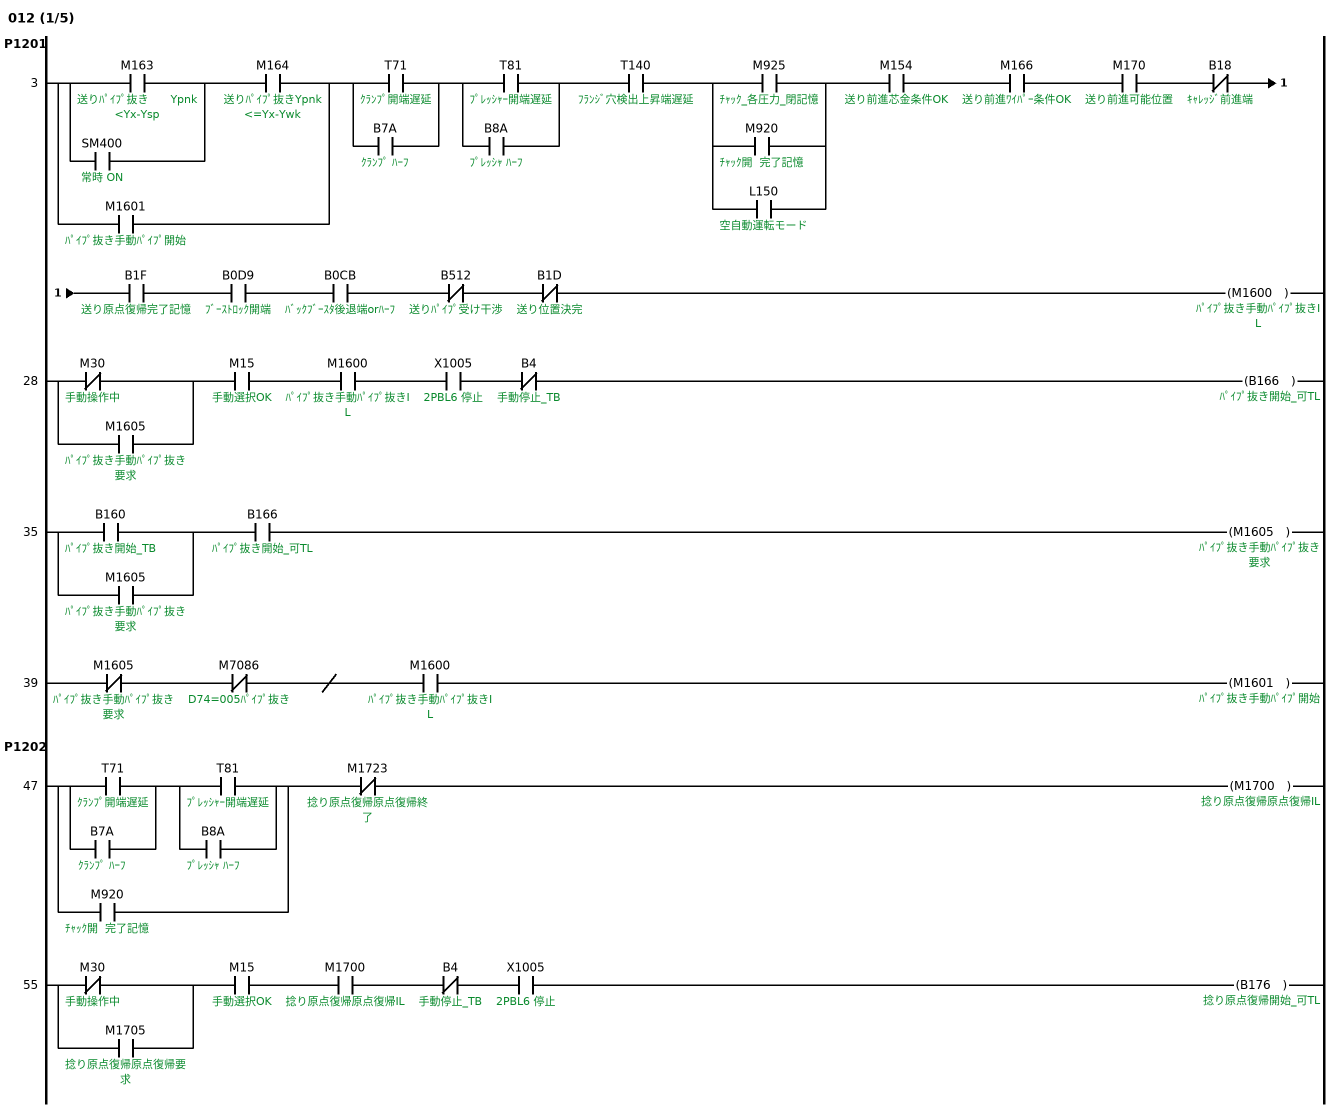
3     LD      M163  ; 送りﾊﾟｲﾌﾟ抜き　　Ypnk<Yx-Ysp
      OR      SM400  ; 常時 ON
      AND     M164  ; 送りﾊﾟｲﾌﾟ抜きYpnk <=Yx-Ywk
      OR      M1601  ; ﾊﾟｲﾌﾟ抜き手動ﾊﾟｲﾌﾟ開始
      LD      T71  ; ｸﾗﾝﾌﾟ開端遅延
      OR      B7A  ; ｸﾗﾝﾌﾟ ﾊｰﾌ
      ANB
      LD      T81  ; ﾌﾟﾚｯｼｬｰ開端遅延
      OR      B8A  ; ﾌﾟﾚｯｼｬ ﾊｰﾌ
      ANB
      AND     T140  ; ﾌﾗﾝｼﾞ穴検出上昇端遅延
      LD      M925  ; ﾁｬｯｸ_各圧力_閉記憶
      OR      M920  ; ﾁｬｯｸ開  完了記憶
      OR      L150  ; 空自動運転モード
      ANB
      AND     M154  ; 送り前進芯金条件OK
      AND     M166  ; 送り前進ﾜｲﾊﾟｰ条件OK
      AND     M170  ; 送り前進可能位置
      ANI     B18  ; ｷｬﾚｯｼﾞ前進端
      AND     B1F  ; 送り原点復帰完了記憶
      AND     B0D9  ; ﾌﾞｰｽﾄﾛｯｸ開端
      AND     B0CB  ; ﾊﾞｯｸﾌﾞｰｽﾀ後退端orﾊｰﾌ
      ANI     B512  ; 送りﾊﾟｲﾌﾟ受け干渉
      ANI     B1D  ; 送り位置決完
      OUT     M1600  ; ﾊﾟｲﾌﾟ抜き手動ﾊﾟｲﾌﾟ抜きIL
28    LDI     M30  ; 手動操作中
      OR      M1605  ; ﾊﾟｲﾌﾟ抜き手動ﾊﾟｲﾌﾟ抜き要求
      AND     M15  ; 手動選択OK
      AND     M1600  ; ﾊﾟｲﾌﾟ抜き手動ﾊﾟｲﾌﾟ抜きIL
      AND     X1005  ; 2PBL6 停止
      ANI     B4  ; 手動停止_TB
      OUT     B166  ; ﾊﾟｲﾌﾟ抜き開始_可TL
35    LD      B160  ; ﾊﾟｲﾌﾟ抜き開始_TB
      OR      M1605  ; ﾊﾟｲﾌﾟ抜き手動ﾊﾟｲﾌﾟ抜き要求
      AND     B166  ; ﾊﾟｲﾌﾟ抜き開始_可TL
      OUT     M1605  ; ﾊﾟｲﾌﾟ抜き手動ﾊﾟｲﾌﾟ抜き要求
39    LDI     M1605  ; ﾊﾟｲﾌﾟ抜き手動ﾊﾟｲﾌﾟ抜き要求
      ANI     M7086  ; D74=005ﾊﾟｲﾌﾟ抜き
      INV
      AND     M1600  ; ﾊﾟｲﾌﾟ抜き手動ﾊﾟｲﾌﾟ抜きIL
      OUT     M1601  ; ﾊﾟｲﾌﾟ抜き手動ﾊﾟｲﾌﾟ開始
; 
      P1202
47    LD      T71  ; ｸﾗﾝﾌﾟ開端遅延
      OR      B7A  ; ｸﾗﾝﾌﾟ ﾊｰﾌ
      LD      T81  ; ﾌﾟﾚｯｼｬｰ開端遅延
      OR      B8A  ; ﾌﾟﾚｯｼｬ ﾊｰﾌ
      ANB
      OR      M920  ; ﾁｬｯｸ開  完了記憶
      ANI     M1723  ; 捻り原点復帰原点復帰終了
      OUT     M1700  ; 捻り原点復帰原点復帰IL
55    LDI     M30  ; 手動操作中
      OR      M1705  ; 捻り原点復帰原点復帰要求
      AND     M15  ; 手動選択OK
      AND     M1700  ; 捻り原点復帰原点復帰IL
      ANI     B4  ; 手動停止_TB
      AND     X1005  ; 2PBL6 停止
      OUT     B176  ; 捻り原点復帰開始_可TL
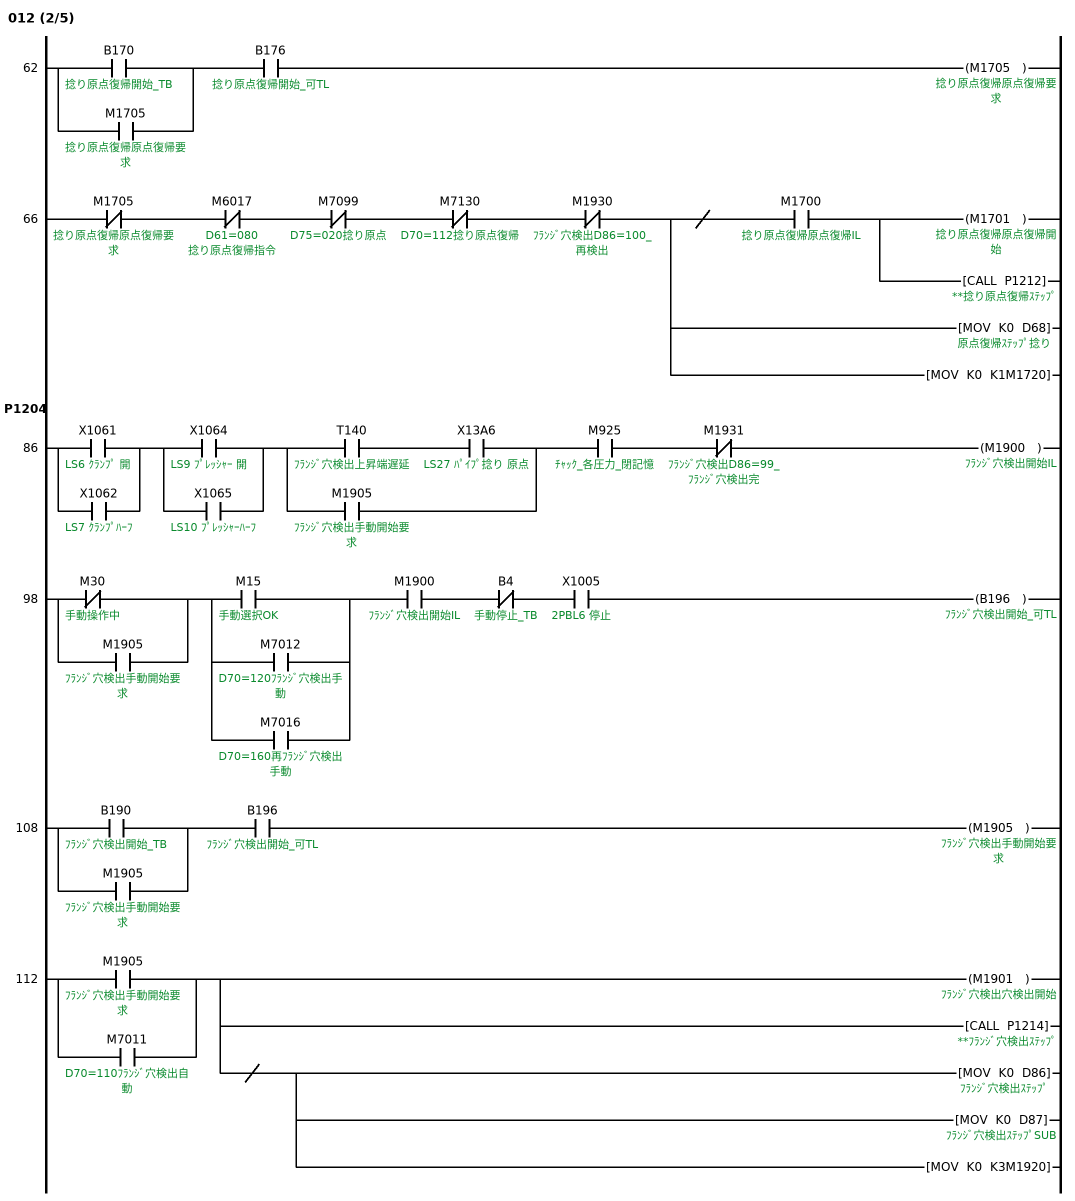
62    LD      B170  ; 捻り原点復帰開始_TB
      OR      M1705  ; 捻り原点復帰原点復帰要求
      AND     B176  ; 捻り原点復帰開始_可TL
      OUT     M1705  ; 捻り原点復帰原点復帰要求
66    LDI     M1705  ; 捻り原点復帰原点復帰要求
      ANI     M6017  ; D61=080 捻り原点復帰指令
      ANI     M7099  ; D75=020捻り原点
      ANI     M7130  ; D70=112捻り原点復帰
      ANI     M1930  ; ﾌﾗﾝｼﾞ穴検出D86=100_再検出
      MPS
      INV
      AND     M1700  ; 捻り原点復帰原点復帰IL
      OUT     M1701  ; 捻り原点復帰原点復帰開始
      CALL    P1212  ; **捻り原点復帰ｽﾃｯﾌﾟ
      MPP
      MOV     K0 D68  ; 原点復帰ｽﾃｯﾌﾟ捻り
      MOV     K0 K1M1720  ; 捻り原点復帰原点復帰逆転
; 
      P1204
86    LD      X1061  ; LS6 ｸﾗﾝﾌﾟ 開
      OR      X1062  ; LS7 ｸﾗﾝﾌﾟﾊｰﾌ
      LD      X1064  ; LS9 ﾌﾟﾚｯｼｬｰ 開
      OR      X1065  ; LS10 ﾌﾟﾚｯｼｬｰﾊｰﾌ
      ANB
      LD      T140  ; ﾌﾗﾝｼﾞ穴検出上昇端遅延
      AND     X13A6  ; LS27 ﾊﾟｲﾌﾟ捻り 原点
      OR      M1905  ; ﾌﾗﾝｼﾞ穴検出手動開始要求
      ANB
      AND     M925  ; ﾁｬｯｸ_各圧力_閉記憶
      ANI     M1931  ; ﾌﾗﾝｼﾞ穴検出D86=99_ﾌﾗﾝｼﾞ穴検出完
      OUT     M1900  ; ﾌﾗﾝｼﾞ穴検出開始IL
98    LDI     M30  ; 手動操作中
      OR      M1905  ; ﾌﾗﾝｼﾞ穴検出手動開始要求
      LD      M15  ; 手動選択OK
      OR      M7012  ; D70=120ﾌﾗﾝｼﾞ穴検出手動
      OR      M7016  ; D70=160再ﾌﾗﾝｼﾞ穴検出手動
      ANB
      AND     M1900  ; ﾌﾗﾝｼﾞ穴検出開始IL
      ANI     B4  ; 手動停止_TB
      AND     X1005  ; 2PBL6 停止
      OUT     B196  ; ﾌﾗﾝｼﾞ穴検出開始_可TL
108   LD      B190  ; ﾌﾗﾝｼﾞ穴検出開始_TB
      OR      M1905  ; ﾌﾗﾝｼﾞ穴検出手動開始要求
      AND     B196  ; ﾌﾗﾝｼﾞ穴検出開始_可TL
      OUT     M1905  ; ﾌﾗﾝｼﾞ穴検出手動開始要求
112   LD      M1905  ; ﾌﾗﾝｼﾞ穴検出手動開始要求
      OR      M7011  ; D70=110ﾌﾗﾝｼﾞ穴検出自動
      OUT     M1901  ; ﾌﾗﾝｼﾞ穴検出穴検出開始
      CALL    P1214  ; **ﾌﾗﾝｼﾞ穴検出ｽﾃｯﾌﾟ
      INV
      MOV     K0 D86  ; ﾌﾗﾝｼﾞ穴検出ｽﾃｯﾌﾟ
      MOV     K0 D87  ; ﾌﾗﾝｼﾞ穴検出ｽﾃｯﾌﾟSUB
      MOV     K0 K3M1920  ; ﾌﾗﾝｼﾞ穴検出D86=010_ﾌﾗﾝｼﾞ穴検下降
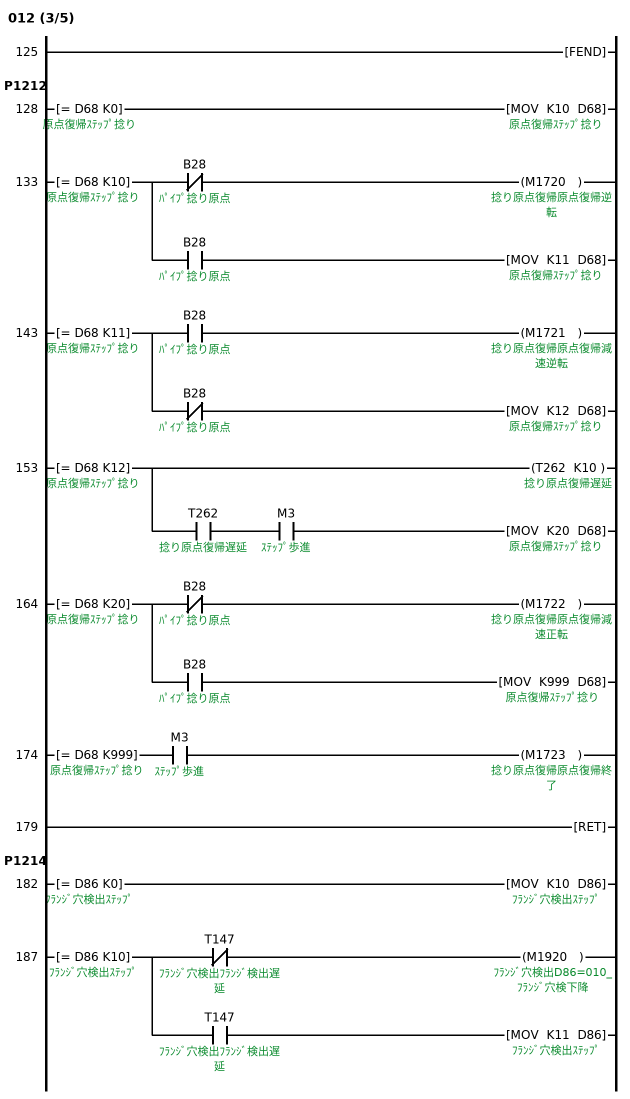
125   FEND
; 
      P1212
128   LD=     D68 K0  ; 原点復帰ｽﾃｯﾌﾟ捻り
      MOV     K10 D68
133   LD=     D68 K10  ; 原点復帰ｽﾃｯﾌﾟ捻り
      MPS
      ANI     B28  ; ﾊﾟｲﾌﾟ捻り原点
      OUT     M1720  ; 捻り原点復帰原点復帰逆転
      MPP
      AND     B28  ; ﾊﾟｲﾌﾟ捻り原点
      MOV     K11 D68
143   LD=     D68 K11  ; 原点復帰ｽﾃｯﾌﾟ捻り
      MPS
      AND     B28  ; ﾊﾟｲﾌﾟ捻り原点
      OUT     M1721  ; 捻り原点復帰原点復帰減速逆転
      MPP
      ANI     B28  ; ﾊﾟｲﾌﾟ捻り原点
      MOV     K12 D68
153   LD=     D68 K12  ; 原点復帰ｽﾃｯﾌﾟ捻り
      OUT     T262 K10  ; 捻り原点復帰遅延
      AND     T262  ; 捻り原点復帰遅延
      AND     M3  ; ｽﾃｯﾌﾟ歩進
      MOV     K20 D68
164   LD=     D68 K20  ; 原点復帰ｽﾃｯﾌﾟ捻り
      MPS
      ANI     B28  ; ﾊﾟｲﾌﾟ捻り原点
      OUT     M1722  ; 捻り原点復帰原点復帰減速正転
      MPP
      AND     B28  ; ﾊﾟｲﾌﾟ捻り原点
      MOV     K999 D68
174   LD=     D68 K999  ; 原点復帰ｽﾃｯﾌﾟ捻り
      AND     M3  ; ｽﾃｯﾌﾟ歩進
      OUT     M1723  ; 捻り原点復帰原点復帰終了
179   RET
; 
      P1214
182   LD=     D86 K0  ; ﾌﾗﾝｼﾞ穴検出ｽﾃｯﾌﾟ
      MOV     K10 D86
187   LD=     D86 K10  ; ﾌﾗﾝｼﾞ穴検出ｽﾃｯﾌﾟ
      MPS
      ANI     T147  ; ﾌﾗﾝｼﾞ穴検出ﾌﾗﾝｼﾞ検出遅延
      OUT     M1920  ; ﾌﾗﾝｼﾞ穴検出D86=010_ﾌﾗﾝｼﾞ穴検下降
      MPP
      AND     T147  ; ﾌﾗﾝｼﾞ穴検出ﾌﾗﾝｼﾞ検出遅延
      MOV     K11 D86
